LIN {X 0,Y 474.155,Z 514.396,A -85,B 0,C 180,E1 20492.017,E2 20492.017} C_VEL
LIN {X 0,Y 475.544,Z 517.886,A -85,B 0,C 180,E1 20491.079,E2 20491.079} C_VEL
LIN {X 0,Y 476.952,Z 519.954,A -85,B 0,C 180,E1 20490.456,E2 20490.456} C_VEL
LIN {X 0,Y 479.191,Z 523.963,A -85,B 0,C 180,E1 20489.394,E2 20489.394} C_VEL
LIN {X 0,Y 481.484,Z 528.373,A -85,B 0,C 180,E1 20488.305,E2 20488.305} C_VEL
LIN {X 0,Y 486.793,Z 538.934,A -85,B 0,C 180,E1 20485.892,E2 20485.892} C_VEL
LIN {X 0,Y 493.143,Z 551.884,A -85,B 0,C 180,E1 20483.213,E2 20483.213} C_VEL
LIN {X 0,Y 495.153,Z 556.027,A -85,B 0,C 180,E1 20482.476,E2 20482.476} C_VEL
LIN {X 0,Y 509.076,Z 575.515,A -85,B 0,C 180,E1 20480.277,E2 20480.277} C_VEL
LIN {X 0,Y 522.792,Z 596.581,A -85,B 0,C 180,E1 20478.273,E2 20478.273} C_VEL
LIN {X 0,Y 527.931,Z 605.432,A -85,B 0,C 180,E1 20477.547,E2 20477.547} C_VEL
LIN {X 0,Y 518.42,Z 845.443,A -85,B 0,C 180,E1 20473.808,E2 20473.808} C_VEL
LIN {X 0,Y 515.244,Z 924.905,A -85,B 0,C 180,E1 20472.535,E2 20472.535} C_VEL
LIN {X 0,Y 513.406,Z 949.561,A -85,B 0,C 180,E1 20471.961,E2 20471.961} C_VEL
LIN {X 0,Y 511.178,Z 973.065,A -85,B 0,C 180,E1 20471.232,E2 20471.232} C_VEL
LIN {X 0,Y 508.452,Z 995.949,A -85,B 0,C 180,E1 20470.313,E2 20470.313} C_VEL
LIN {X 0,Y 505.435,Z 1018.304,A -85,B 0,C 180,E1 20469.227,E2 20469.227} C_VEL
LIN {X 0,Y 502.044,Z 1040.134,A -85,B 0,C 180,E1 20467.936,E2 20467.936} C_VEL
LIN {X 0,Y 498.656,Z 1060.29,A -85,B 0,C 180,E1 20466.549,E2 20466.549} C_VEL
LIN {X 0,Y 494.89,Z 1080.931,A -85,B 0,C 180,E1 20464.873,E2 20464.873} C_VEL
LIN {X 0,Y 491.266,Z 1100.34,A -85,B 0,C 180,E1 20463.055,E2 20463.055} C_VEL
LIN {X 0,Y 487.78,Z 1118.193,A -85,B 0,C 180,E1 20461.101,E2 20461.101} C_VEL
LIN {X 0,Y 484.436,Z 1135.567,A -85,B 0,C 180,E1 20458.937,E2 20458.937} C_VEL
LIN {X 0,Y 481.445,Z 1151.258,A -85,B 0,C 180,E1 20456.653,E2 20456.653} C_VEL
LIN {X 0,Y 478.757,Z 1166.255,A -85,B 0,C 180,E1 20454.163,E2 20454.163} C_VEL
LIN {X 0,Y 476.612,Z 1179.063,A -85,B 0,C 180,E1 20451.662,E2 20451.662} C_VEL
LIN {X 0,Y 474.889,Z 1190.823,A -85,B 0,C 180,E1 20449.023,E2 20449.023} C_VEL
LIN {X 0,Y 473.606,Z 1200.885,A -85,B 0,C 180,E1 20446.307,E2 20446.307} C_VEL
LIN {X 0,Y 472.768,Z 1209.435,A -85,B 0,C 180,E1 20443.577,E2 20443.577} C_VEL
LIN {X 0,Y 472.242,Z 1216.419,A -85,B 0,C 180,E1 20440.738,E2 20440.738} C_VEL
LIN {X 0,Y 472.032,Z 1221.191,A -85,B 0,C 180,E1 20438.282,E2 20438.282} C_VEL
LIN {X 0,Y 471.92,Z 1225.242,A -85,B 0,C 180,E1 20435.349,E2 20435.349} C_VEL
LIN {X 0,Y 471.913,Z 1227.184,A -85,B 0,C 180,E1 20433.036,E2 20433.036} C_VEL
LIN {X 0,Y 471.916,Z 1228.071,A -85,B 0,C 180,E1 20430.728,E2 20430.728} C_VEL
LIN {X 0,Y 471.93,Z 1227.822,A -85,B 0,C 180,E1 20428.057,E2 20428.057} C_VEL
LIN {X 0,Y 471.933,Z 1225.961,A -85,B 0,C 180,E1 20425.382,E2 20425.382} C_VEL
LIN {X 0,Y 471.984,Z 1223.075,A -85,B 0,C 180,E1 20422.942,E2 20422.942} C_VEL
LIN {X 0,Y 472.159,Z 1218.019,A -85,B 0,C 180,E1 20420,E2 20420} C_VEL
LIN {X 0,Y 472.543,Z 1212,A -85,B 0,C 180,E1 20417.412,E2 20417.412} C_VEL
LIN {X 0,Y 473.256,Z 1204.234,A -85,B 0,C 180,E1 20414.687,E2 20414.687} C_VEL
LIN {X 0,Y 474.378,Z 1194.449,A -85,B 0,C 180,E1 20411.919,E2 20411.919} C_VEL
LIN {X 0,Y 475.903,Z 1183.735,A -85,B 0,C 180,E1 20409.331,E2 20409.331} C_VEL
LIN {X 0,Y 477.969,Z 1170.754,A -85,B 0,C 180,E1 20406.69,E2 20406.69} C_VEL
LIN {X 0,Y 480.439,Z 1156.789,A -85,B 0,C 180,E1 20404.218,E2 20404.218} C_VEL
LIN {X 0,Y 483.33,Z 1141.174,A -85,B 0,C 180,E1 20401.858,E2 20401.858} C_VEL
LIN {X 0,Y 486.577,Z 1124.421,A -85,B 0,C 180,E1 20399.635,E2 20399.635} C_VEL
LIN {X 0,Y 490.009,Z 1106.609,A -85,B 0,C 180,E1 20397.614,E2 20397.614} C_VEL
LIN {X 0,Y 493.65,Z 1087.708,A -85,B 0,C 180,E1 20395.732,E2 20395.732} C_VEL
LIN {X 0,Y 497.245,Z 1067.846,A -85,B 0,C 180,E1 20394.045,E2 20394.045} C_VEL
LIN {X 0,Y 500.924,Z 1046.802,A -85,B 0,C 180,E1 20392.498,E2 20392.498} C_VEL
LIN {X 0,Y 504.252,Z 1025.704,A -85,B 0,C 180,E1 20391.196,E2 20391.196} C_VEL
LIN {X 0,Y 507.471,Z 1003.563,A -85,B 0,C 180,E1 20390.036,E2 20390.036} C_VEL
LIN {X 0,Y 510.126,Z 981.826,A -85,B 0,C 180,E1 20389.107,E2 20389.107} C_VEL
LIN {X 0,Y 512.636,Z 958.481,A -85,B 0,C 180,E1 20388.297,E2 20388.297} C_VEL
LIN {X 0,Y 514.535,Z 935.049,A -85,B 0,C 180,E1 20387.69,E2 20387.69} C_VEL
LIN {X 0,Y 515.919,Z 910.67,A -85,B 0,C 180,E1 20387.223,E2 20387.223} C_VEL
LIN {X 0,Y 525.461,Z 664.98,A -85,B 0,C 180,E1 20383.375,E2 20383.375} C_VEL
LIN {X 0,Y 527.752,Z 604.829,A -85,B 0,C 180,E1 20382.433,E2 20382.433} C_VEL
LIN {X 0,Y 514.53,Z 583.673,A -85,B 0,C 180,E1 20380.552,E2 20380.552} C_VEL
LIN {X 0,Y 500.408,Z 563.192,A -85,B 0,C 180,E1 20378.402,E2 20378.402} C_VEL
LIN {X 0,Y 494.767,Z 555.412,A -85,B 0,C 180,E1 20377.467,E2 20377.467} C_VEL
LIN {X 0,Y 488.441,Z 542.064,A -85,B 0,C 180,E1 20374.829,E2 20374.829} C_VEL
LIN {X 0,Y 483.454,Z 532.413,A -85,B 0,C 180,E1 20372.671,E2 20372.671} C_VEL
LIN {X 0,Y 480.951,Z 527.653,A -85,B 0,C 180,E1 20371.531,E2 20371.531} C_VEL
LIN {X 0,Y 478.491,Z 523.082,A -85,B 0,C 180,E1 20370.378,E2 20370.378} C_VEL
LIN {X 0,Y 476.323,Z 518.832,A -85,B 0,C 180,E1 20369.282,E2 20369.282} C_VEL
LIN {X 0,Y 474.366,Z 515.411,A -85,B 0,C 180,E1 20368.312,E2 20368.312} C_VEL
LIN {X 0,Y 474.133,Z 514.262,A -85,B 0,C 180,E1 20367.916,E2 20367.916} C_VEL
LIN {X 0,Y 474.098,Z 514.151,A -85,B 0,C 180,E1 20364.284,E2 20364.284} C_VEL
LIN {X 0,Y 474.071,Z 514.151,A -85,B 0,C 180,E1 20360.753,E2 20360.753} C_VEL
LIN {X 0,Y 474.09,Z 514.148,A -85,B 0,C 180,E1 20357.174,E2 20357.174} C_VEL
LIN {X 0,Y 474.118,Z 514.152,A -85,B 0,C 180,E1 20353.663,E2 20353.663} C_VEL
LIN {X 0,Y 474.088,Z 514.176,A -85,B 0,C 180,E1 20350.082,E2 20350.082} C_VEL
LIN {X 0,Y 474.077,Z 514.166,A -85,B 0,C 180,E1 20346.418,E2 20346.418} C_VEL
LIN {X 0,Y 474.094,Z 514.146,A -85,B 0,C 180,E1 20342.78,E2 20342.78} C_VEL
LIN {X 0,Y 474.116,Z 514.142,A -85,B 0,C 180,E1 20339.275,E2 20339.275} C_VEL
LIN {X 0,Y 474.09,Z 514.163,A -85,B 0,C 180,E1 20335.645,E2 20335.645} C_VEL
LIN {X 0,Y 474.082,Z 514.178,A -85,B 0,C 180,E1 20331.998,E2 20331.998} C_VEL
LIN {X 0,Y 474.102,Z 514.154,A -85,B 0,C 180,E1 20328.442,E2 20328.442} C_VEL
LIN {X 0,Y 474.115,Z 514.143,A -85,B 0,C 180,E1 20324.84,E2 20324.84} C_VEL
LIN {X 0,Y 474.093,Z 514.147,A -85,B 0,C 180,E1 20321.251,E2 20321.251} C_VEL
LIN {X 0,Y 474.086,Z 514.154,A -85,B 0,C 180,E1 20317.689,E2 20317.689} C_VEL
LIN {X 0,Y 474.111,Z 514.156,A -85,B 0,C 180,E1 20314.115,E2 20314.115} C_VEL
LIN {X 0,Y 474.127,Z 514.429,A -85,B 0,C 180,E1 20311.467,E2 20311.467} C_VEL
LIN {X 0,Y 475.735,Z 518.072,A -85,B 0,C 180,E1 20310.471,E2 20310.471} C_VEL
LIN {X 0,Y 476.903,Z 519.937,A -85,B 0,C 180,E1 20309.927,E2 20309.927} C_VEL
LIN {X 0,Y 478.881,Z 523.608,A -85,B 0,C 180,E1 20308.954,E2 20308.954} C_VEL
LIN {X 0,Y 482.172,Z 530.174,A -85,B 0,C 180,E1 20307.341,E2 20307.341} C_VEL
LIN {X 0,Y 484.724,Z 535.255,A -85,B 0,C 180,E1 20306.154,E2 20306.154} C_VEL
LIN {X 0,Y 489.09,Z 544.038,A -85,B 0,C 180,E1 20304.218,E2 20304.218} C_VEL
LIN {X 0,Y 494.758,Z 556.102,A -85,B 0,C 180,E1 20301.799,E2 20301.799} C_VEL
LIN {X 0,Y 501.517,Z 571.621,A -85,B 0,C 180,E1 20299.009,E2 20299.009} C_VEL
LIN {X 0,Y 508.454,Z 589.192,A -85,B 0,C 180,E1 20296.194,E2 20296.194} C_VEL
LIN {X 0,Y 513.484,Z 603.577,A -85,B 0,C 180,E1 20294.117,E2 20294.117} C_VEL
LIN {X 0,Y 510.099,Z 627.117,A -85,B 0,C 180,E1 20292.145,E2 20292.145} C_VEL
LIN {X 0,Y 518.572,Z 680.793,A -85,B 0,C 180,E1 20290.232,E2 20290.232} C_VEL
LIN {X 0,Y 521.342,Z 700.88,A -85,B 0,C 180,E1 20289.597,E2 20289.597} C_VEL
LIN {X 0,Y 514.32,Z 951.65,A -85,B 0,C 180,E1 20286.124,E2 20286.124} C_VEL
LIN {X 0,Y 512.707,Z 973.976,A -85,B 0,C 180,E1 20285.653,E2 20285.653} C_VEL
LIN {X 0,Y 510.551,Z 995.541,A -85,B 0,C 180,E1 20285.016,E2 20285.016} C_VEL
LIN {X 0,Y 508.063,Z 1015.095,A -85,B 0,C 180,E1 20284.251,E2 20284.251} C_VEL
LIN {X 0,Y 504.852,Z 1036.457,A -85,B 0,C 180,E1 20283.203,E2 20283.203} C_VEL
LIN {X 0,Y 501.504,Z 1055.972,A -85,B 0,C 180,E1 20282.028,E2 20282.028} C_VEL
LIN {X 0,Y 497.867,Z 1074.515,A -85,B 0,C 180,E1 20280.671,E2 20280.671} C_VEL
LIN {X 0,Y 493.994,Z 1093.026,A -85,B 0,C 180,E1 20279.063,E2 20279.063} C_VEL
LIN {X 0,Y 490.378,Z 1109.28,A -85,B 0,C 180,E1 20277.39,E2 20277.39} C_VEL
LIN {X 0,Y 486.854,Z 1124.477,A -85,B 0,C 180,E1 20275.549,E2 20275.549} C_VEL
LIN {X 0,Y 486.127,Z 1127.636,A -85,B 0,C 180,E1 20275.13,E2 20275.13} C_VEL
LIN {X 0,Y 484.064,Z 1132.744,A -85,B 0,C 180,E1 20274.483,E2 20274.483} C_VEL
LIN {X 0,Y 475.596,Z 1145.16,A -85,B 0,C 180,E1 20272.883,E2 20272.883} C_VEL
LIN {X 0,Y 473.58,Z 1149.608,A -85,B 0,C 180,E1 20272.155,E2 20272.155} C_VEL
LIN {X 0,Y 470.739,Z 1161.868,A -85,B 0,C 180,E1 20269.784,E2 20269.784} C_VEL
LIN {X 0,Y 468.375,Z 1172.626,A -85,B 0,C 180,E1 20267.261,E2 20267.261} C_VEL
LIN {X 0,Y 466.516,Z 1182.255,A -85,B 0,C 180,E1 20264.522,E2 20264.522} C_VEL
LIN {X 0,Y 465.325,Z 1189.709,A -85,B 0,C 180,E1 20261.904,E2 20261.904} C_VEL
LIN {X 0,Y 464.56,Z 1195.655,A -85,B 0,C 180,E1 20259.164,E2 20259.164} C_VEL
LIN {X 0,Y 464.143,Z 1200.188,A -85,B 0,C 180,E1 20256.307,E2 20256.307} C_VEL
LIN {X 0,Y 464.002,Z 1202.847,A -85,B 0,C 180,E1 20253.707,E2 20253.707} C_VEL
LIN {X 0,Y 463.961,Z 1204.118,A -85,B 0,C 180,E1 20250.988,E2 20250.988} C_VEL
LIN {X 0,Y 463.962,Z 1204.008,A -85,B 0,C 180,E1 20248.271,E2 20248.271} C_VEL
LIN {X 0,Y 464.03,Z 1202.291,A -85,B 0,C 180,E1 20245.551,E2 20245.551} C_VEL
LIN {X 0,Y 464.238,Z 1198.967,A -85,B 0,C 180,E1 20242.7,E2 20242.7} C_VEL
LIN {X 0,Y 464.702,Z 1194.401,A -85,B 0,C 180,E1 20240.088,E2 20240.088} C_VEL
LIN {X 0,Y 465.569,Z 1187.959,A -85,B 0,C 180,E1 20237.346,E2 20237.346} C_VEL
LIN {X 0,Y 466.914,Z 1180.215,A -85,B 0,C 180,E1 20234.728,E2 20234.728} C_VEL
LIN {X 0,Y 468.827,Z 1170.537,A -85,B 0,C 180,E1 20232.115,E2 20232.115} C_VEL
LIN {X 0,Y 471.404,Z 1158.887,A -85,B 0,C 180,E1 20229.515,E2 20229.515} C_VEL
LIN {X 0,Y 474.37,Z 1146.429,A -85,B 0,C 180,E1 20227.181,E2 20227.181} C_VEL
LIN {X 0,Y 477.553,Z 1133.278,A -85,B 0,C 180,E1 20225.113,E2 20225.113} C_VEL
LIN {X 0,Y 481.473,Z 1117.091,A -85,B 0,C 180,E1 20222.949,E2 20222.949} C_VEL
LIN {X 0,Y 485.362,Z 1100.85,A -85,B 0,C 180,E1 20221.109,E2 20221.109} C_VEL
LIN {X 0,Y 489.163,Z 1083.804,A -85,B 0,C 180,E1 20219.491,E2 20219.491} C_VEL
LIN {X 0,Y 493.259,Z 1064.206,A -85,B 0,C 180,E1 20217.921,E2 20217.921} C_VEL
LIN {X 0,Y 496.963,Z 1044.87,A -85,B 0,C 180,E1 20216.634,E2 20216.634} C_VEL
LIN {X 0,Y 500.265,Z 1024.901,A -85,B 0,C 180,E1 20215.555,E2 20215.555} C_VEL
LIN {X 0,Y 503.312,Z 1003.371,A -85,B 0,C 180,E1 20214.614,E2 20214.614} C_VEL
LIN {X 0,Y 505.699,Z 982.724,A -85,B 0,C 180,E1 20213.917,E2 20213.917} C_VEL
LIN {X 0,Y 507.619,Z 960.502,A -85,B 0,C 180,E1 20213.375,E2 20213.375} C_VEL
LIN {X 0,Y 508.783,Z 936.875,A -85,B 0,C 180,E1 20212.979,E2 20212.979} C_VEL
LIN {X 0,Y 515.475,Z 700.609,A -85,B 0,C 180,E1 20209.68,E2 20209.68} C_VEL
LIN {X 0,Y 507.716,Z 648.72,A -85,B 0,C 180,E1 20207.879,E2 20207.879} C_VEL
LIN {X 0,Y 504.105,Z 625.337,A -85,B 0,C 180,E1 20206.976,E2 20206.976} C_VEL
LIN {X 0,Y 506.962,Z 606.936,A -85,B 0,C 180,E1 20205.399,E2 20205.399} C_VEL
LIN {X 0,Y 500.415,Z 588.775,A -85,B 0,C 180,E1 20202.669,E2 20202.669} C_VEL
LIN {X 0,Y 493.848,Z 572.457,A -85,B 0,C 180,E1 20199.929,E2 20199.929} C_VEL
LIN {X 0,Y 487.537,Z 558.088,A -85,B 0,C 180,E1 20197.23,E2 20197.23} C_VEL
LIN {X 0,Y 482.013,Z 546.324,A -85,B 0,C 180,E1 20194.771,E2 20194.771} C_VEL
LIN {X 0,Y 477.796,Z 537.861,A -85,B 0,C 180,E1 20192.821,E2 20192.821} C_VEL
LIN {X 0,Y 475.073,Z 532.675,A -85,B 0,C 180,E1 20191.529,E2 20191.529} C_VEL
LIN {X 0,Y 473.555,Z 529.451,A -85,B 0,C 180,E1 20190.729,E2 20190.729} C_VEL
LIN {X 0,Y 471.63,Z 525.759,A -85,B 0,C 180,E1 20189.742,E2 20189.742} C_VEL
LIN {X 0,Y 469.026,Z 521.007,A -85,B 0,C 180,E1 20188.386,E2 20188.386} C_VEL
LIN {X 0,Y 466.326,Z 516.083,A -85,B 0,C 180,E1 20186.881,E2 20186.881} C_VEL
LIN {X 0,Y 466.157,Z 515.237,A -85,B 0,C 180,E1 20186.497,E2 20186.497} C_VEL
LIN {X 0,Y 466.147,Z 515.137,A -85,B 0,C 180,E1 20182.732,E2 20182.732} C_VEL
LIN {X 0,Y 466.173,Z 515.132,A -85,B 0,C 180,E1 20179.158,E2 20179.158} C_VEL
LIN {X 0,Y 466.171,Z 515.136,A -85,B 0,C 180,E1 20175.552,E2 20175.552} C_VEL
LIN {X 0,Y 466.142,Z 515.158,A -85,B 0,C 180,E1 20172.009,E2 20172.009} C_VEL
LIN {X 0,Y 466.144,Z 515.166,A -85,B 0,C 180,E1 20168.263,E2 20168.263} C_VEL
LIN {X 0,Y 466.166,Z 515.14,A -85,B 0,C 180,E1 20164.675,E2 20164.675} C_VEL
LIN {X 0,Y 466.173,Z 515.129,A -85,B 0,C 180,E1 20160.983,E2 20160.983} C_VEL
LIN {X 0,Y 466.14,Z 515.141,A -85,B 0,C 180,E1 20157.418,E2 20157.418} C_VEL
LIN {X 0,Y 466.139,Z 515.162,A -85,B 0,C 180,E1 20153.719,E2 20153.719} C_VEL
LIN {X 0,Y 466.159,Z 515.157,A -85,B 0,C 180,E1 20150.119,E2 20150.119} C_VEL
LIN {X 0,Y 466.177,Z 515.137,A -85,B 0,C 180,E1 20146.48,E2 20146.48} C_VEL
LIN {X 0,Y 466.141,Z 515.135,A -85,B 0,C 180,E1 20142.91,E2 20142.91} C_VEL
LIN {X 0,Y 466.131,Z 515.138,A -85,B 0,C 180,E1 20139.264,E2 20139.264} C_VEL
LIN {X 0,Y 466.155,Z 515.139,A -85,B 0,C 180,E1 20135.68,E2 20135.68} C_VEL
LIN {X 0,Y 466.204,Z 515.444,A -85,B 0,C 180,E1 20133.681,E2 20133.681} C_VEL
LIN {X 0,Y 467.491,Z 518.71,A -85,B 0,C 180,E1 20132.76,E2 20132.76} C_VEL
LIN {X 0,Y 469.06,Z 520.891,A -85,B 0,C 180,E1 20132.032,E2 20132.032} C_VEL
LIN {X 0,Y 470.968,Z 524.611,A -85,B 0,C 180,E1 20131.006,E2 20131.006} C_VEL
LIN {X 0,Y 472.301,Z 527.272,A -85,B 0,C 180,E1 20130.304,E2 20130.304} C_VEL
LIN {X 0,Y 474.398,Z 531.003,A -85,B 0,C 180,E1 20129.307,E2 20129.307} C_VEL
LIN {X 0,Y 477.153,Z 536.384,A -85,B 0,C 180,E1 20127.983,E2 20127.983} C_VEL
LIN {X 0,Y 481.197,Z 544.202,A -85,B 0,C 180,E1 20126.159,E2 20126.159} C_VEL
LIN {X 0,Y 487.509,Z 557.043,A -85,B 0,C 180,E1 20123.502,E2 20123.502} C_VEL
LIN {X 0,Y 501.063,Z 575.927,A -85,B 0,C 180,E1 20121.255,E2 20121.255} C_VEL
LIN {X 0,Y 513.716,Z 594.998,A -85,B 0,C 180,E1 20119.323,E2 20119.323} C_VEL
LIN {X 0,Y 522.067,Z 608.776,A -85,B 0,C 180,E1 20118.108,E2 20118.108} C_VEL
LIN {X 0,Y 512.25,Z 848.274,A -85,B 0,C 180,E1 20114.346,E2 20114.346} C_VEL
LIN {X 0,Y 509.051,Z 925.38,A -85,B 0,C 180,E1 20113.099,E2 20113.099} C_VEL
LIN {X 0,Y 507.158,Z 949.918,A -85,B 0,C 180,E1 20112.522,E2 20112.522} C_VEL
LIN {X 0,Y 504.866,Z 973.275,A -85,B 0,C 180,E1 20111.791,E2 20111.791} C_VEL
LIN {X 0,Y 502.065,Z 996.036,A -85,B 0,C 180,E1 20110.87,E2 20110.87} C_VEL
LIN {X 0,Y 498.862,Z 1018.969,A -85,B 0,C 180,E1 20109.744,E2 20109.744} C_VEL
LIN {X 0,Y 495.344,Z 1040.705,A -85,B 0,C 180,E1 20108.44,E2 20108.44} C_VEL
LIN {X 0,Y 491.751,Z 1061.312,A -85,B 0,C 180,E1 20107.002,E2 20107.002} C_VEL
LIN {X 0,Y 487.845,Z 1081.773,A -85,B 0,C 180,E1 20105.308,E2 20105.308} C_VEL
LIN {X 0,Y 483.989,Z 1101.508,A -85,B 0,C 180,E1 20103.421,E2 20103.421} C_VEL
LIN {X 0,Y 480.46,Z 1118.817,A -85,B 0,C 180,E1 20101.489,E2 20101.489} C_VEL
LIN {X 0,Y 476.999,Z 1136.02,A -85,B 0,C 180,E1 20099.305,E2 20099.305} C_VEL
LIN {X 0,Y 473.864,Z 1151.706,A -85,B 0,C 180,E1 20096.978,E2 20096.978} C_VEL
LIN {X 0,Y 471.06,Z 1166.601,A -85,B 0,C 180,E1 20094.45,E2 20094.45} C_VEL
LIN {X 0,Y 468.825,Z 1179.341,A -85,B 0,C 180,E1 20091.912,E2 20091.912} C_VEL
LIN {X 0,Y 466.954,Z 1191.423,A -85,B 0,C 180,E1 20089.124,E2 20089.124} C_VEL
LIN {X 0,Y 465.674,Z 1201.048,A -85,B 0,C 180,E1 20086.464,E2 20086.464} C_VEL
LIN {X 0,Y 464.796,Z 1209.535,A -85,B 0,C 180,E1 20083.688,E2 20083.688} C_VEL
LIN {X 0,Y 464.261,Z 1216.335,A -85,B 0,C 180,E1 20080.856,E2 20080.856} C_VEL
LIN {X 0,Y 464.035,Z 1221.186,A -85,B 0,C 180,E1 20078.3,E2 20078.3} C_VEL
LIN {X 0,Y 463.924,Z 1225.031,A -85,B 0,C 180,E1 20075.441,E2 20075.441} C_VEL
LIN {X 0,Y 463.916,Z 1226.978,A -85,B 0,C 180,E1 20073.089,E2 20073.089} C_VEL
LIN {X 0,Y 463.919,Z 1227.866,A -85,B 0,C 180,E1 20070.741,E2 20070.741} C_VEL
LIN {X 0,Y 463.933,Z 1227.617,A -85,B 0,C 180,E1 20068.024,E2 20068.024} C_VEL
LIN {X 0,Y 463.931,Z 1225.75,A -85,B 0,C 180,E1 20065.302,E2 20065.302} C_VEL
LIN {X 0,Y 463.985,Z 1223.027,A -85,B 0,C 180,E1 20062.944,E2 20062.944} C_VEL
LIN {X 0,Y 464.155,Z 1218.322,A -85,B 0,C 180,E1 20060.077,E2 20060.077} C_VEL
LIN {X 0,Y 464.563,Z 1212.076,A -85,B 0,C 180,E1 20057.319,E2 20057.319} C_VEL
LIN {X 0,Y 465.263,Z 1204.723,A -85,B 0,C 180,E1 20054.673,E2 20054.673} C_VEL
LIN {X 0,Y 466.404,Z 1195.252,A -85,B 0,C 180,E1 20051.89,E2 20051.89} C_VEL
LIN {X 0,Y 467.871,Z 1185.251,A -85,B 0,C 180,E1 20049.4,E2 20049.4} C_VEL
LIN {X 0,Y 470.103,Z 1171.867,A -85,B 0,C 180,E1 20046.564,E2 20046.564} C_VEL
LIN {X 0,Y 472.378,Z 1159.368,A -85,B 0,C 180,E1 20044.284,E2 20044.284} C_VEL
LIN {X 0,Y 475.658,Z 1142.549,A -85,B 0,C 180,E1 20041.637,E2 20041.637} C_VEL
LIN {X 0,Y 478.798,Z 1126.91,A -85,B 0,C 180,E1 20039.506,E2 20039.506} C_VEL
LIN {X 0,Y 482.55,Z 1108.439,A -85,B 0,C 180,E1 20037.333,E2 20037.333} C_VEL
LIN {X 0,Y 486.038,Z 1091.007,A -85,B 0,C 180,E1 20035.548,E2 20035.548} C_VEL
LIN {X 0,Y 490.049,Z 1070.067,A -85,B 0,C 180,E1 20033.703,E2 20033.703} C_VEL
LIN {X 0,Y 493.756,Z 1049.73,A -85,B 0,C 180,E1 20032.165,E2 20032.165} C_VEL
LIN {X 0,Y 497.354,Z 1028.058,A -85,B 0,C 180,E1 20030.783,E2 20030.783} C_VEL
LIN {X 0,Y 500.502,Z 1007.339,A -85,B 0,C 180,E1 20029.665,E2 20029.665} C_VEL
LIN {X 0,Y 503.594,Z 983.594,A -85,B 0,C 180,E1 20028.612,E2 20028.612} C_VEL
LIN {X 0,Y 506.006,Z 961.948,A -85,B 0,C 180,E1 20027.839,E2 20027.839} C_VEL
LIN {X 0,Y 508.183,Z 937.31,A -85,B 0,C 180,E1 20027.169,E2 20027.169} C_VEL
LIN {X 0,Y 509.549,Z 915.033,A -85,B 0,C 180,E1 20026.725,E2 20026.725} C_VEL
LIN {X 0,Y 519.396,Z 671.122,A -85,B 0,C 180,E1 20022.865,E2 20022.865} C_VEL
LIN {X 0,Y 521.884,Z 608.216,A -85,B 0,C 180,E1 20021.872,E2 20021.872} C_VEL
LIN {X 0,Y 508.399,Z 586.776,A -85,B 0,C 180,E1 20019.897,E2 20019.897} C_VEL
LIN {X 0,Y 494.504,Z 566.61,A -85,B 0,C 180,E1 20017.71,E2 20017.71} C_VEL
LIN {X 0,Y 487.167,Z 556.44,A -85,B 0,C 180,E1 20016.435,E2 20016.435} C_VEL
LIN {X 0,Y 480.604,Z 542.941,A -85,B 0,C 180,E1 20013.601,E2 20013.601} C_VEL
LIN {X 0,Y 475.803,Z 533.692,A -85,B 0,C 180,E1 20011.411,E2 20011.411} C_VEL
LIN {X 0,Y 473.231,Z 528.939,A -85,B 0,C 180,E1 20010.19,E2 20010.19} C_VEL
LIN {X 0,Y 471.072,Z 524.729,A -85,B 0,C 180,E1 20009.083,E2 20009.083} C_VEL
LIN {X 0,Y 469.122,Z 521.117,A -85,B 0,C 180,E1 20008.07,E2 20008.07} C_VEL
LIN {X 0,Y 468.152,Z 519.517,A -85,B 0,C 180,E1 20007.584,E2 20007.584} C_VEL
LIN {X 0,Y 466.386,Z 516.358,A -85,B 0,C 180,E1 20006.621,E2 20006.621} C_VEL
LIN {X 0,Y 466.18,Z 515.248,A -85,B 0,C 180,E1 20006.222,E2 20006.222} C_VEL
LIN {X 0,Y 466.137,Z 515.165,A -85,B 0,C 180,E1 20002.713,E2 20002.713} C_VEL
LIN {X 0,Y 466.143,Z 515.168,A -85,B 0,C 180,E1 19999.029,E2 19999.029} C_VEL
LIN {X 0,Y 466.179,Z 515.15,A -85,B 0,C 180,E1 19995.424,E2 19995.424} C_VEL
LIN {X 0,Y 466.167,Z 515.136,A -85,B 0,C 180,E1 19991.757,E2 19991.757} C_VEL
LIN {X 0,Y 466.139,Z 515.13,A -85,B 0,C 180,E1 19988.139,E2 19988.139} C_VEL
LIN {X 0,Y 466.139,Z 515.138,A -85,B 0,C 180,E1 19984.429,E2 19984.429} C_VEL
LIN {X 0,Y 466.162,Z 515.159,A -85,B 0,C 180,E1 19980.737,E2 19980.737} C_VEL
LIN {X 0,Y 466.175,Z 515.157,A -85,B 0,C 180,E1 19977.049,E2 19977.049} C_VEL
LIN {X 0,Y 466.167,Z 515.136,A -85,B 0,C 180,E1 19973.349,E2 19973.349} C_VEL
LIN {X 0,Y 466.142,Z 515.133,A -85,B 0,C 180,E1 19969.744,E2 19969.744} C_VEL
LIN {X 0,Y 466.152,Z 515.14,A -85,B 0,C 180,E1 19966.099,E2 19966.099} C_VEL
LIN {X 0,Y 466.177,Z 515.154,A -85,B 0,C 180,E1 19962.525,E2 19962.525} C_VEL
LIN {X 0,Y 466.175,Z 515.164,A -85,B 0,C 180,E1 19958.879,E2 19958.879} C_VEL
LIN {X 0,Y 466.149,Z 515.163,A -85,B 0,C 180,E1 19955.274,E2 19955.274} C_VEL
LIN {X 0,Y 466.197,Z 515.449,A -85,B 0,C 180,E1 19953.151,E2 19953.151} C_VEL
LIN {X 0,Y 467.784,Z 519.045,A -85,B 0,C 180,E1 19952.088,E2 19952.088} C_VEL
LIN {X 0,Y 469.02,Z 520.979,A -85,B 0,C 180,E1 19951.475,E2 19951.475} C_VEL
LIN {X 0,Y 471.172,Z 524.818,A -85,B 0,C 180,E1 19950.366,E2 19950.366} C_VEL
LIN {X 0,Y 473.564,Z 529.455,A -85,B 0,C 180,E1 19949.131,E2 19949.131} C_VEL
LIN {X 0,Y 478.643,Z 539.359,A -85,B 0,C 180,E1 19946.673,E2 19946.673} C_VEL
LIN {X 0,Y 485.077,Z 552.741,A -85,B 0,C 180,E1 19943.73,E2 19943.73} C_VEL
LIN {X 0,Y 491.581,Z 567.183,A -85,B 0,C 180,E1 19940.909,E2 19940.909} C_VEL
LIN {X 0,Y 498.329,Z 583.494,A -85,B 0,C 180,E1 19938.075,E2 19938.075} C_VEL
LIN {X 0,Y 505.021,Z 601.388,A -85,B 0,C 180,E1 19935.297,E2 19935.297} C_VEL
LIN {X 0,Y 506.908,Z 606.859,A -85,B 0,C 180,E1 19934.506,E2 19934.506} C_VEL
LIN {X 0,Y 504.045,Z 626.234,A -85,B 0,C 180,E1 19932.87,E2 19932.87} C_VEL
LIN {X 0,Y 512.128,Z 678.026,A -85,B 0,C 180,E1 19930.975,E2 19930.975} C_VEL
LIN {X 0,Y 515.471,Z 702.355,A -85,B 0,C 180,E1 19930.185,E2 19930.185} C_VEL
LIN {X 0,Y 508.157,Z 951.353,A -85,B 0,C 180,E1 19926.7,E2 19926.7} C_VEL
LIN {X 0,Y 506.503,Z 973.594,A -85,B 0,C 180,E1 19926.229,E2 19926.229} C_VEL
LIN {X 0,Y 504.374,Z 994.496,A -85,B 0,C 180,E1 19925.614,E2 19925.614} C_VEL
LIN {X 0,Y 501.603,Z 1015.5,A -85,B 0,C 180,E1 19924.787,E2 19924.787} C_VEL
LIN {X 0,Y 498.256,Z 1036.893,A -85,B 0,C 180,E1 19923.723,E2 19923.723} C_VEL
LIN {X 0,Y 494.75,Z 1056.62,A -85,B 0,C 180,E1 19922.518,E2 19922.518} C_VEL
LIN {X 0,Y 490.991,Z 1075.05,A -85,B 0,C 180,E1 19921.148,E2 19921.148} C_VEL
LIN {X 0,Y 486.978,Z 1093.469,A -85,B 0,C 180,E1 19919.522,E2 19919.522} C_VEL
LIN {X 0,Y 483.176,Z 1109.95,A -85,B 0,C 180,E1 19917.801,E2 19917.801} C_VEL
LIN {X 0,Y 479.356,Z 1125.728,A -85,B 0,C 180,E1 19915.845,E2 19915.845} C_VEL
LIN {X 0,Y 475.927,Z 1139.912,A -85,B 0,C 180,E1 19913.789,E2 19913.789} C_VEL
LIN {X 0,Y 473.58,Z 1149.608,A -85,B 0,C 180,E1 19912.155,E2 19912.155} C_VEL
LIN {X 0,Y 471.604,Z 1154.028,A -85,B 0,C 180,E1 19911.407,E2 19911.407} C_VEL
LIN {X 0,Y 463.475,Z 1164.458,A -85,B 0,C 180,E1 19909.551,E2 19909.551} C_VEL
LIN {X 0,Y 461.698,Z 1168.191,A -85,B 0,C 180,E1 19908.743,E2 19908.743} C_VEL
LIN {X 0,Y 459.564,Z 1177.934,A -85,B 0,C 180,E1 19906.17,E2 19906.17} C_VEL
LIN {X 0,Y 457.944,Z 1186.584,A -85,B 0,C 180,E1 19903.382,E2 19903.382} C_VEL
LIN {X 0,Y 456.948,Z 1193.11,A -85,B 0,C 180,E1 19900.719,E2 19900.719} C_VEL
LIN {X 0,Y 456.344,Z 1198.249,A -85,B 0,C 180,E1 19897.934,E2 19897.934} C_VEL
LIN {X 0,Y 456.069,Z 1201.882,A -85,B 0,C 180,E1 19895.157,E2 19895.157} C_VEL
LIN {X 0,Y 455.978,Z 1203.86,A -85,B 0,C 180,E1 19892.388,E2 19892.388} C_VEL
LIN {X 0,Y 455.955,Z 1204.424,A -85,B 0,C 180,E1 19889.497,E2 19889.497} C_VEL
LIN {X 0,Y 455.988,Z 1203.528,A -85,B 0,C 180,E1 19886.858,E2 19886.858} C_VEL
LIN {X 0,Y 456.122,Z 1200.966,A -85,B 0,C 180,E1 19883.96,E2 19883.96} C_VEL
LIN {X 0,Y 456.488,Z 1197.021,A -85,B 0,C 180,E1 19881.18,E2 19881.18} C_VEL
LIN {X 0,Y 457.2,Z 1191.321,A -85,B 0,C 180,E1 19878.393,E2 19878.393} C_VEL
LIN {X 0,Y 458.487,Z 1183.56,A -85,B 0,C 180,E1 19875.476,E2 19875.476} C_VEL
LIN {X 0,Y 460.268,Z 1174.731,A -85,B 0,C 180,E1 19872.816,E2 19872.816} C_VEL
LIN {X 0,Y 462.567,Z 1164.411,A -85,B 0,C 180,E1 19870.294,E2 19870.294} C_VEL
LIN {X 0,Y 465.552,Z 1152.084,A -85,B 0,C 180,E1 19867.772,E2 19867.772} C_VEL
LIN {X 0,Y 468.993,Z 1138.508,A -85,B 0,C 180,E1 19865.435,E2 19865.435} C_VEL
LIN {X 0,Y 472.647,Z 1124.053,A -85,B 0,C 180,E1 19863.354,E2 19863.354} C_VEL
LIN {X 0,Y 476.825,Z 1107.25,A -85,B 0,C 180,E1 19861.302,E2 19861.302} C_VEL
LIN {X 0,Y 480.844,Z 1090.624,A -85,B 0,C 180,E1 19859.58,E2 19859.58} C_VEL
LIN {X 0,Y 484.749,Z 1073.043,A -85,B 0,C 180,E1 19858.058,E2 19858.058} C_VEL
LIN {X 0,Y 488.655,Z 1054.163,A -85,B 0,C 180,E1 19856.675,E2 19856.675} C_VEL
LIN {X 0,Y 492.092,Z 1035.425,A -85,B 0,C 180,E1 19855.537,E2 19855.537} C_VEL
LIN {X 0,Y 495.364,Z 1015.075,A -85,B 0,C 180,E1 19854.529,E2 19854.529} C_VEL
LIN {X 0,Y 498.22,Z 994.116,A -85,B 0,C 180,E1 19853.699,E2 19853.699} C_VEL
LIN {X 0,Y 500.452,Z 972.815,A -85,B 0,C 180,E1 19853.072,E2 19853.072} C_VEL
LIN {X 0,Y 502.159,Z 949.965,A -85,B 0,C 180,E1 19852.593,E2 19852.593} C_VEL
LIN {X 0,Y 509.687,Z 702.178,A -85,B 0,C 180,E1 19849.083,E2 19849.083} C_VEL
LIN {X 0,Y 502.03,Z 649.959,A -85,B 0,C 180,E1 19847.235,E2 19847.235} C_VEL
LIN {X 0,Y 498.128,Z 624.609,A -85,B 0,C 180,E1 19846.244,E2 19846.244} C_VEL
LIN {X 0,Y 500.37,Z 610.512,A -85,B 0,C 180,E1 19845.024,E2 19845.024} C_VEL
LIN {X 0,Y 494.157,Z 593.11,A -85,B 0,C 180,E1 19842.361,E2 19842.361} C_VEL
LIN {X 0,Y 487.628,Z 576.713,A -85,B 0,C 180,E1 19839.559,E2 19839.559} C_VEL
LIN {X 0,Y 481.52,Z 562.728,A -85,B 0,C 180,E1 19836.879,E2 19836.879} C_VEL
LIN {X 0,Y 476.017,Z 550.946,A -85,B 0,C 180,E1 19834.363,E2 19834.363} C_VEL
LIN {X 0,Y 470.741,Z 540.046,A -85,B 0,C 180,E1 19831.788,E2 19831.788} C_VEL
LIN {X 0,Y 467.697,Z 534.485,A -85,B 0,C 180,E1 19830.301,E2 19830.301} C_VEL
LIN {X 0,Y 465.608,Z 530.334,A -85,B 0,C 180,E1 19829.175,E2 19829.175} C_VEL
LIN {X 0,Y 463.096,Z 525.617,A -85,B 0,C 180,E1 19827.799,E2 19827.799} C_VEL
LIN {X 0,Y 461.136,Z 521.934,A -85,B 0,C 180,E1 19826.67,E2 19826.67} C_VEL
LIN {X 0,Y 458.395,Z 517.091,A -85,B 0,C 180,E1 19825.035,E2 19825.035} C_VEL
LIN {X 0,Y 458.215,Z 516.214,A -85,B 0,C 180,E1 19824.632,E2 19824.632} C_VEL
LIN {X 0,Y 458.226,Z 516.153,A -85,B 0,C 180,E1 19820.949,E2 19820.949} C_VEL
LIN {X 0,Y 458.239,Z 516.144,A -85,B 0,C 180,E1 19817.263,E2 19817.263} C_VEL
LIN {X 0,Y 458.232,Z 516.132,A -85,B 0,C 180,E1 19813.502,E2 19813.502} C_VEL
LIN {X 0,Y 458.205,Z 516.123,A -85,B 0,C 180,E1 19809.8,E2 19809.8} C_VEL
LIN {X 0,Y 458.199,Z 516.122,A -85,B 0,C 180,E1 19806.138,E2 19806.138} C_VEL
LIN {X 0,Y 458.22,Z 516.135,A -85,B 0,C 180,E1 19802.501,E2 19802.501} C_VEL
LIN {X 0,Y 458.241,Z 516.153,A -85,B 0,C 180,E1 19798.875,E2 19798.875} C_VEL
LIN {X 0,Y 458.215,Z 516.135,A -85,B 0,C 180,E1 19795.118,E2 19795.118} C_VEL
LIN {X 0,Y 458.191,Z 516.122,A -85,B 0,C 180,E1 19791.593,E2 19791.593} C_VEL
LIN {X 0,Y 458.215,Z 516.124,A -85,B 0,C 180,E1 19788.036,E2 19788.036} C_VEL
LIN {X 0,Y 458.244,Z 516.134,A -85,B 0,C 180,E1 19784.432,E2 19784.432} C_VEL
LIN {X 0,Y 458.213,Z 516.15,A -85,B 0,C 180,E1 19780.761,E2 19780.761} C_VEL
LIN {X 0,Y 458.194,Z 516.156,A -85,B 0,C 180,E1 19777.142,E2 19777.142} C_VEL
LIN {X 0,Y 458.258,Z 516.481,A -85,B 0,C 180,E1 19775.531,E2 19775.531} C_VEL
LIN {X 0,Y 459.675,Z 519.837,A -85,B 0,C 180,E1 19774.488,E2 19774.488} C_VEL
LIN {X 0,Y 461.146,Z 521.871,A -85,B 0,C 180,E1 19773.747,E2 19773.747} C_VEL
LIN {X 0,Y 463.102,Z 525.636,A -85,B 0,C 180,E1 19772.62,E2 19772.62} C_VEL
LIN {X 0,Y 464.052,Z 527.265,A -85,B 0,C 180,E1 19772.123,E2 19772.123} C_VEL
LIN {X 0,Y 466.862,Z 532.602,A -85,B 0,C 180,E1 19770.629,E2 19770.629} C_VEL
LIN {X 0,Y 469.319,Z 537.289,A -85,B 0,C 180,E1 19769.39,E2 19769.39} C_VEL
LIN {X 0,Y 471.86,Z 542.221,A -85,B 0,C 180,E1 19768.154,E2 19768.154} C_VEL
LIN {X 0,Y 476.093,Z 550.656,A -85,B 0,C 180,E1 19766.182,E2 19766.182} C_VEL
LIN {X 0,Y 479.907,Z 558.307,A -85,B 0,C 180,E1 19764.568,E2 19764.568} C_VEL
LIN {X 0,Y 492.546,Z 575.495,A -85,B 0,C 180,E1 19762.372,E2 19762.372} C_VEL
LIN {X 0,Y 506.218,Z 595.701,A -85,B 0,C 180,E1 19760.192,E2 19760.192} C_VEL
LIN {X 0,Y 516.258,Z 612.041,A -85,B 0,C 180,E1 19758.684,E2 19758.684} C_VEL
LIN {X 0,Y 506.127,Z 851.124,A -85,B 0,C 180,E1 19754.898,E2 19754.898} C_VEL
LIN {X 0,Y 502.917,Z 925.749,A -85,B 0,C 180,E1 19753.679,E2 19753.679} C_VEL
LIN {X 0,Y 500.966,Z 950.215,A -85,B 0,C 180,E1 19753.098,E2 19753.098} C_VEL
LIN {X 0,Y 498.594,Z 973.605,A -85,B 0,C 180,E1 19752.361,E2 19752.361} C_VEL
LIN {X 0,Y 495.677,Z 996.511,A -85,B 0,C 180,E1 19751.424,E2 19751.424} C_VEL
LIN {X 0,Y 492.389,Z 1019.228,A -85,B 0,C 180,E1 19750.297,E2 19750.297} C_VEL
LIN {X 0,Y 488.905,Z 1040.01,A -85,B 0,C 180,E1 19749.042,E2 19749.042} C_VEL
LIN {X 0,Y 485.176,Z 1060.687,A -85,B 0,C 180,E1 19747.589,E2 19747.589} C_VEL
LIN {X 0,Y 481.109,Z 1081.253,A -85,B 0,C 180,E1 19745.878,E2 19745.878} C_VEL
LIN {X 0,Y 477.172,Z 1100.614,A -85,B 0,C 180,E1 19744.019,E2 19744.019} C_VEL
LIN {X 0,Y 473.271,Z 1118.925,A -85,B 0,C 180,E1 19741.953,E2 19741.953} C_VEL
LIN {X 0,Y 469.667,Z 1136.099,A -85,B 0,C 180,E1 19739.737,E2 19739.737} C_VEL
LIN {X 0,Y 466.459,Z 1151.362,A -85,B 0,C 180,E1 19737.442,E2 19737.442} C_VEL
LIN {X 0,Y 463.65,Z 1165.621,A -85,B 0,C 180,E1 19735.003,E2 19735.003} C_VEL
LIN {X 0,Y 461.251,Z 1178.44,A -85,B 0,C 180,E1 19732.428,E2 19732.428} C_VEL
LIN {X 0,Y 459.31,Z 1190.168,A -85,B 0,C 180,E1 19729.719,E2 19729.719} C_VEL
LIN {X 0,Y 457.849,Z 1200.365,A -85,B 0,C 180,E1 19726.885,E2 19726.885} C_VEL
LIN {X 0,Y 456.918,Z 1208.568,A -85,B 0,C 180,E1 19724.187,E2 19724.187} C_VEL
LIN {X 0,Y 456.312,Z 1215.691,A -85,B 0,C 180,E1 19721.246,E2 19721.246} C_VEL
LIN {X 0,Y 456.063,Z 1220.53,A -85,B 0,C 180,E1 19718.701,E2 19718.701} C_VEL
LIN {X 0,Y 455.934,Z 1224.701,A -85,B 0,C 180,E1 19715.663,E2 19715.663} C_VEL
LIN {X 0,Y 455.919,Z 1226.772,A -85,B 0,C 180,E1 19713.143,E2 19713.143} C_VEL
LIN {X 0,Y 455.922,Z 1227.662,A -85,B 0,C 180,E1 19710.754,E2 19710.754} C_VEL
LIN {X 0,Y 455.935,Z 1227.411,A -85,B 0,C 180,E1 19707.989,E2 19707.989} C_VEL
LIN {X 0,Y 455.929,Z 1225.54,A -85,B 0,C 180,E1 19705.22,E2 19705.22} C_VEL
LIN {X 0,Y 455.98,Z 1222.811,A -85,B 0,C 180,E1 19702.82,E2 19702.82} C_VEL
LIN {X 0,Y 456.168,Z 1218.093,A -85,B 0,C 180,E1 19699.901,E2 19699.901} C_VEL
LIN {X 0,Y 456.609,Z 1211.837,A -85,B 0,C 180,E1 19697.094,E2 19697.094} C_VEL
LIN {X 0,Y 457.358,Z 1204.473,A -85,B 0,C 180,E1 19694.401,E2 19694.401} C_VEL
LIN {X 0,Y 458.601,Z 1194.798,A -85,B 0,C 180,E1 19691.521,E2 19691.521} C_VEL
LIN {X 0,Y 460.158,Z 1184.774,A -85,B 0,C 180,E1 19688.991,E2 19688.991} C_VEL
LIN {X 0,Y 462.517,Z 1171.427,A -85,B 0,C 180,E1 19686.13,E2 19686.13} C_VEL
LIN {X 0,Y 464.9,Z 1159.038,A -85,B 0,C 180,E1 19683.839,E2 19683.839} C_VEL
LIN {X 0,Y 468.171,Z 1143.053,A -85,B 0,C 180,E1 19681.28,E2 19681.28} C_VEL
LIN {X 0,Y 471.435,Z 1127.476,A -85,B 0,C 180,E1 19679.119,E2 19679.119} C_VEL
LIN {X 0,Y 475.455,Z 1108.559,A -85,B 0,C 180,E1 19676.855,E2 19676.855} C_VEL
LIN {X 0,Y 479.085,Z 1091.147,A -85,B 0,C 180,E1 19675.048,E2 19675.048} C_VEL
LIN {X 0,Y 483.185,Z 1070.594,A -85,B 0,C 180,E1 19673.211,E2 19673.211} C_VEL
LIN {X 0,Y 486.971,Z 1050.602,A -85,B 0,C 180,E1 19671.679,E2 19671.679} C_VEL
LIN {X 0,Y 490.834,Z 1028.29,A -85,B 0,C 180,E1 19670.235,E2 19670.235} C_VEL
LIN {X 0,Y 494.089,Z 1007.594,A -85,B 0,C 180,E1 19669.107,E2 19669.107} C_VEL
LIN {X 0,Y 497.285,Z 983.886,A -85,B 0,C 180,E1 19668.046,E2 19668.046} C_VEL
LIN {X 0,Y 499.741,Z 962.554,A -85,B 0,C 180,E1 19667.277,E2 19667.277} C_VEL
LIN {X 0,Y 502.018,Z 937.672,A -85,B 0,C 180,E1 19666.592,E2 19666.592} C_VEL
LIN {X 0,Y 503.419,Z 915.54,A -85,B 0,C 180,E1 19666.146,E2 19666.146} C_VEL
LIN {X 0,Y 513.606,Z 671.851,A -85,B 0,C 180,E1 19662.258,E2 19662.258} C_VEL
LIN {X 0,Y 516.062,Z 611.643,A -85,B 0,C 180,E1 19661.298,E2 19661.298} C_VEL
LIN {X 0,Y 503.03,Z 590.912,A -85,B 0,C 180,E1 19659.334,E2 19659.334} C_VEL
LIN {X 0,Y 489.157,Z 570.851,A -85,B 0,C 180,E1 19657.086,E2 19657.086} C_VEL
LIN {X 0,Y 479.666,Z 557.927,A -85,B 0,C 180,E1 19655.409,E2 19655.409} C_VEL
LIN {X 0,Y 473.146,Z 544.537,A -85,B 0,C 180,E1 19652.464,E2 19652.464} C_VEL
LIN {X 0,Y 468.261,Z 535.198,A -85,B 0,C 180,E1 19650.119,E2 19650.119} C_VEL
LIN {X 0,Y 465.771,Z 530.551,A -85,B 0,C 180,E1 19648.856,E2 19648.856} C_VEL
LIN {X 0,Y 463.21,Z 525.755,A -85,B 0,C 180,E1 19647.482,E2 19647.482} C_VEL
LIN {X 0,Y 461.233,Z 522.176,A -85,B 0,C 180,E1 19646.386,E2 19646.386} C_VEL
LIN {X 0,Y 460.341,Z 520.625,A -85,B 0,C 180,E1 19645.886,E2 19645.886} C_VEL
LIN {X 0,Y 458.422,Z 517.268,A -85,B 0,C 180,E1 19644.758,E2 19644.758} C_VEL
LIN {X 0,Y 458.228,Z 516.229,A -85,B 0,C 180,E1 19644.357,E2 19644.357} C_VEL
LIN {X 0,Y 458.194,Z 516.127,A -85,B 0,C 180,E1 19640.837,E2 19640.837} C_VEL
LIN {X 0,Y 458.218,Z 516.123,A -85,B 0,C 180,E1 19637.264,E2 19637.264} C_VEL
LIN {X 0,Y 458.24,Z 516.127,A -85,B 0,C 180,E1 19633.631,E2 19633.631} C_VEL
LIN {X 0,Y 458.218,Z 516.146,A -85,B 0,C 180,E1 19629.927,E2 19629.927} C_VEL
LIN {X 0,Y 458.202,Z 516.146,A -85,B 0,C 180,E1 19626.264,E2 19626.264} C_VEL
LIN {X 0,Y 458.203,Z 516.127,A -85,B 0,C 180,E1 19622.501,E2 19622.501} C_VEL
LIN {X 0,Y 458.235,Z 516.117,A -85,B 0,C 180,E1 19619,E2 19619} C_VEL
LIN {X 0,Y 458.225,Z 516.131,A -85,B 0,C 180,E1 19615.369,E2 19615.369} C_VEL
LIN {X 0,Y 458.209,Z 516.155,A -85,B 0,C 180,E1 19611.719,E2 19611.719} C_VEL
LIN {X 0,Y 458.209,Z 516.142,A -85,B 0,C 180,E1 19608.035,E2 19608.035} C_VEL
LIN {X 0,Y 458.233,Z 516.124,A -85,B 0,C 180,E1 19604.431,E2 19604.431} C_VEL
LIN {X 0,Y 458.235,Z 516.121,A -85,B 0,C 180,E1 19600.762,E2 19600.762} C_VEL
LIN {X 0,Y 458.216,Z 516.125,A -85,B 0,C 180,E1 19597.144,E2 19597.144} C_VEL
LIN {X 0,Y 458.262,Z 516.437,A -85,B 0,C 180,E1 19595,E2 19595} C_VEL
LIN {X 0,Y 459.92,Z 520.147,A -85,B 0,C 180,E1 19593.811,E2 19593.811} C_VEL
LIN {X 0,Y 461.125,Z 521.877,A -85,B 0,C 180,E1 19593.191,E2 19593.191} C_VEL
LIN {X 0,Y 463.269,Z 525.838,A -85,B 0,C 180,E1 19591.973,E2 19591.973} C_VEL
LIN {X 0,Y 466.537,Z 532.128,A -85,B 0,C 180,E1 19590.183,E2 19590.183} C_VEL
LIN {X 0,Y 469.477,Z 537.933,A -85,B 0,C 180,E1 19588.652,E2 19588.652} C_VEL
LIN {X 0,Y 473.273,Z 545.203,A -85,B 0,C 180,E1 19586.825,E2 19586.825} C_VEL
LIN {X 0,Y 479.378,Z 557.983,A -85,B 0,C 180,E1 19583.971,E2 19583.971} C_VEL
LIN {X 0,Y 485.791,Z 572.423,A -85,B 0,C 180,E1 19581.114,E2 19581.114} C_VEL
LIN {X 0,Y 492.449,Z 588.754,A -85,B 0,C 180,E1 19578.242,E2 19578.242} C_VEL
LIN {X 0,Y 498.968,Z 606.458,A -85,B 0,C 180,E1 19575.463,E2 19575.463} C_VEL
LIN {X 0,Y 500.321,Z 610.568,A -85,B 0,C 180,E1 19574.866,E2 19574.866} C_VEL
LIN {X 0,Y 498.068,Z 625.287,A -85,B 0,C 180,E1 19573.617,E2 19573.617} C_VEL
LIN {X 0,Y 505.938,Z 676.469,A -85,B 0,C 180,E1 19571.696,E2 19571.696} C_VEL
LIN {X 0,Y 509.657,Z 703.677,A -85,B 0,C 180,E1 19570.788,E2 19570.788} C_VEL
LIN {X 0,Y 502.045,Z 951.04,A -85,B 0,C 180,E1 19567.292,E2 19567.292} C_VEL
LIN {X 0,Y 500.335,Z 973.387,A -85,B 0,C 180,E1 19566.815,E2 19566.815} C_VEL
LIN {X 0,Y 498.207,Z 993.756,A -85,B 0,C 180,E1 19566.215,E2 19566.215} C_VEL
LIN {X 0,Y 495.393,Z 1014.486,A -85,B 0,C 180,E1 19565.398,E2 19565.398} C_VEL
LIN {X 0,Y 491.942,Z 1035.963,A -85,B 0,C 180,E1 19564.334,E2 19564.334} C_VEL
LIN {X 0,Y 488.329,Z 1055.686,A -85,B 0,C 180,E1 19563.127,E2 19563.127} C_VEL
LIN {X 0,Y 484.441,Z 1074.226,A -85,B 0,C 180,E1 19561.747,E2 19561.747} C_VEL
LIN {X 0,Y 480.431,Z 1092.123,A -85,B 0,C 180,E1 19560.172,E2 19560.172} C_VEL
LIN {X 0,Y 476.467,Z 1108.609,A -85,B 0,C 180,E1 19558.448,E2 19558.448} C_VEL
LIN {X 0,Y 472.456,Z 1124.676,A -85,B 0,C 180,E1 19556.462,E2 19556.462} C_VEL
LIN {X 0,Y 468.724,Z 1139.475,A -85,B 0,C 180,E1 19554.311,E2 19554.311} C_VEL
LIN {X 0,Y 465.469,Z 1152.345,A -85,B 0,C 180,E1 19552.081,E2 19552.081} C_VEL
LIN {X 0,Y 462.519,Z 1164.547,A -85,B 0,C 180,E1 19549.577,E2 19549.577} C_VEL
LIN {X 0,Y 461.698,Z 1168.191,A -85,B 0,C 180,E1 19548.743,E2 19548.743} C_VEL
LIN {X 0,Y 459.97,Z 1171.808,A -85,B 0,C 180,E1 19547.916,E2 19547.916} C_VEL
LIN {X 0,Y 452.022,Z 1180.641,A -85,B 0,C 180,E1 19545.698,E2 19545.698} C_VEL
LIN {X 0,Y 450.781,Z 1183.06,A -85,B 0,C 180,E1 19544.928,E2 19544.928} C_VEL
LIN {X 0,Y 449.46,Z 1190.458,A -85,B 0,C 180,E1 19542.201,E2 19542.201} C_VEL
LIN {X 0,Y 448.62,Z 1196.333,A -85,B 0,C 180,E1 19539.364,E2 19539.364} C_VEL
LIN {X 0,Y 448.165,Z 1200.758,A -85,B 0,C 180,E1 19536.405,E2 19536.405} C_VEL
LIN {X 0,Y 448.006,Z 1203.475,A -85,B 0,C 180,E1 19533.583,E2 19533.583} C_VEL
LIN {X 0,Y 447.966,Z 1204.569,A -85,B 0,C 180,E1 19530.767,E2 19530.767} C_VEL
LIN {X 0,Y 447.976,Z 1204.306,A -85,B 0,C 180,E1 19527.953,E2 19527.953} C_VEL
LIN {X 0,Y 448.048,Z 1202.598,A -85,B 0,C 180,E1 19525.264,E2 19525.264} C_VEL
LIN {X 0,Y 448.308,Z 1199.197,A -85,B 0,C 180,E1 19522.31,E2 19522.31} C_VEL
LIN {X 0,Y 448.846,Z 1194.593,A -85,B 0,C 180,E1 19519.605,E2 19519.605} C_VEL
LIN {X 0,Y 449.851,Z 1188.077,A -85,B 0,C 180,E1 19516.766,E2 19516.766} C_VEL
LIN {X 0,Y 451.399,Z 1180.133,A -85,B 0,C 180,E1 19514.02,E2 19514.02} C_VEL
LIN {X 0,Y 453.53,Z 1170.544,A -85,B 0,C 180,E1 19511.357,E2 19511.357} C_VEL
LIN {X 0,Y 456.242,Z 1159.432,A -85,B 0,C 180,E1 19508.802,E2 19508.802} C_VEL
LIN {X 0,Y 459.53,Z 1146.797,A -85,B 0,C 180,E1 19506.356,E2 19506.356} C_VEL
LIN {X 0,Y 463.138,Z 1133.097,A -85,B 0,C 180,E1 19504.145,E2 19504.145} C_VEL
LIN {X 0,Y 467.277,Z 1117.329,A -85,B 0,C 180,E1 19501.987,E2 19501.987} C_VEL
LIN {X 0,Y 471.458,Z 1101.141,A -85,B 0,C 180,E1 19500.107,E2 19500.107} C_VEL
LIN {X 0,Y 475.585,Z 1083.918,A -85,B 0,C 180,E1 19498.433,E2 19498.433} C_VEL
LIN {X 0,Y 479.939,Z 1064.552,A -85,B 0,C 180,E1 19496.848,E2 19496.848} C_VEL
LIN {X 0,Y 483.776,Z 1045.825,A -85,B 0,C 180,E1 19495.572,E2 19495.572} C_VEL
LIN {X 0,Y 487.225,Z 1026.567,A -85,B 0,C 180,E1 19494.496,E2 19494.496} C_VEL
LIN {X 0,Y 490.344,Z 1006.652,A -85,B 0,C 180,E1 19493.581,E2 19493.581} C_VEL
LIN {X 0,Y 493.014,Z 985.298,A -85,B 0,C 180,E1 19492.827,E2 19492.827} C_VEL
LIN {X 0,Y 495.257,Z 962.152,A -85,B 0,C 180,E1 19492.227,E2 19492.227} C_VEL
LIN {X 0,Y 496.562,Z 939.63,A -85,B 0,C 180,E1 19491.825,E2 19491.825} C_VEL
LIN {X 0,Y 503.906,Z 703.383,A -85,B 0,C 180,E1 19488.459,E2 19488.459} C_VEL
LIN {X 0,Y 496.392,Z 651.176,A -85,B 0,C 180,E1 19486.576,E2 19486.576} C_VEL
LIN {X 0,Y 492.253,Z 623.646,A -85,B 0,C 180,E1 19485.477,E2 19485.477} C_VEL
LIN {X 0,Y 493.793,Z 614.102,A -85,B 0,C 180,E1 19484.64,E2 19484.64} C_VEL
LIN {X 0,Y 487.678,Z 596.828,A -85,B 0,C 180,E1 19481.944,E2 19481.944} C_VEL
LIN {X 0,Y 481.391,Z 580.827,A -85,B 0,C 180,E1 19479.156,E2 19479.156} C_VEL
LIN {X 0,Y 474.741,Z 565.495,A -85,B 0,C 180,E1 19476.138,E2 19476.138} C_VEL
LIN {X 0,Y 469.148,Z 553.681,A -85,B 0,C 180,E1 19473.505,E2 19473.505} C_VEL
LIN {X 0,Y 464.84,Z 544.963,A -85,B 0,C 180,E1 19471.358,E2 19471.358} C_VEL
LIN {X 0,Y 462.416,Z 540.306,A -85,B 0,C 180,E1 19470.11,E2 19470.11} C_VEL
LIN {X 0,Y 460.342,Z 536.185,A -85,B 0,C 180,E1 19468.971,E2 19468.971} C_VEL
LIN {X 0,Y 457.851,Z 531.5,A -85,B 0,C 180,E1 19467.58,E2 19467.58} C_VEL
LIN {X 0,Y 455.255,Z 526.716,A -85,B 0,C 180,E1 19466.057,E2 19466.057} C_VEL
LIN {X 0,Y 453.252,Z 522.875,A -85,B 0,C 180,E1 19464.781,E2 19464.781} C_VEL
LIN {X 0,Y 450.599,Z 518.525,A -85,B 0,C 180,E1 19463.127,E2 19463.127} C_VEL
LIN {X 0,Y 450.28,Z 517.219,A -85,B 0,C 180,E1 19462.592,E2 19462.592} C_VEL
LIN {X 0,Y 450.283,Z 517.109,A -85,B 0,C 180,E1 19458.918,E2 19458.918} C_VEL
LIN {X 0,Y 450.301,Z 517.107,A -85,B 0,C 180,E1 19455.19,E2 19455.19} C_VEL
LIN {X 0,Y 450.285,Z 517.119,A -85,B 0,C 180,E1 19451.528,E2 19451.528} C_VEL
LIN {X 0,Y 450.264,Z 517.145,A -85,B 0,C 180,E1 19447.914,E2 19447.914} C_VEL
LIN {X 0,Y 450.265,Z 517.13,A -85,B 0,C 180,E1 19444.203,E2 19444.203} C_VEL
LIN {X 0,Y 450.292,Z 517.109,A -85,B 0,C 180,E1 19440.509,E2 19440.509} C_VEL
LIN {X 0,Y 450.292,Z 517.106,A -85,B 0,C 180,E1 19436.818,E2 19436.818} C_VEL
LIN {X 0,Y 450.274,Z 517.12,A -85,B 0,C 180,E1 19433.113,E2 19433.113} C_VEL
LIN {X 0,Y 450.26,Z 517.143,A -85,B 0,C 180,E1 19429.379,E2 19429.379} C_VEL
LIN {X 0,Y 450.257,Z 517.138,A -85,B 0,C 180,E1 19425.598,E2 19425.598} C_VEL
LIN {X 0,Y 450.287,Z 517.118,A -85,B 0,C 180,E1 19422.022,E2 19422.022} C_VEL
LIN {X 0,Y 450.303,Z 517.119,A -85,B 0,C 180,E1 19418.234,E2 19418.234} C_VEL
LIN {X 0,Y 450.358,Z 517.697,A -85,B 0,C 180,E1 19417.55,E2 19417.55} C_VEL
LIN {X 0,Y 452.013,Z 521.166,A -85,B 0,C 180,E1 19416.315,E2 19416.315} C_VEL
LIN {X 0,Y 453.26,Z 522.834,A -85,B 0,C 180,E1 19415.637,E2 19415.637} C_VEL
LIN {X 0,Y 455.02,Z 526.401,A -85,B 0,C 180,E1 19414.488,E2 19414.488} C_VEL
LIN {X 0,Y 456.178,Z 528.208,A -85,B 0,C 180,E1 19413.86,E2 19413.86} C_VEL
LIN {X 0,Y 458.17,Z 531.882,A -85,B 0,C 180,E1 19412.723,E2 19412.723} C_VEL
LIN {X 0,Y 461.762,Z 538.714,A -85,B 0,C 180,E1 19410.764,E2 19410.764} C_VEL
LIN {X 0,Y 466.114,Z 546.958,A -85,B 0,C 180,E1 19408.582,E2 19408.582} C_VEL
LIN {X 0,Y 472.348,Z 559.437,A -85,B 0,C 180,E1 19405.694,E2 19405.694} C_VEL
LIN {X 0,Y 483.973,Z 575.174,A -85,B 0,C 180,E1 19403.56,E2 19403.56} C_VEL
LIN {X 0,Y 496.841,Z 593.705,A -85,B 0,C 180,E1 19401.4,E2 19401.4} C_VEL
LIN {X 0,Y 509.694,Z 614.008,A -85,B 0,C 180,E1 19399.393,E2 19399.393} C_VEL
LIN {X 0,Y 510.48,Z 615.79,A -85,B 0,C 180,E1 19399.265,E2 19399.265} C_VEL
LIN {X 0,Y 500.041,Z 854.249,A -85,B 0,C 180,E1 19395.458,E2 19395.458} C_VEL
LIN {X 0,Y 496.839,Z 926.092,A -85,B 0,C 180,E1 19394.274,E2 19394.274} C_VEL
LIN {X 0,Y 494.825,Z 950.562,A -85,B 0,C 180,E1 19393.688,E2 19393.688} C_VEL
LIN {X 0,Y 492.376,Z 973.951,A -85,B 0,C 180,E1 19392.945,E2 19392.945} C_VEL
LIN {X 0,Y 489.38,Z 996.682,A -85,B 0,C 180,E1 19392.007,E2 19392.007} C_VEL
LIN {X 0,Y 485.965,Z 1019.493,A -85,B 0,C 180,E1 19390.865,E2 19390.865} C_VEL
LIN {X 0,Y 482.303,Z 1040.544,A -85,B 0,C 180,E1 19389.579,E2 19389.579} C_VEL
LIN {X 0,Y 478.345,Z 1061.718,A -85,B 0,C 180,E1 19388.07,E2 19388.07} C_VEL
LIN {X 0,Y 474.134,Z 1082.111,A -85,B 0,C 180,E1 19386.34,E2 19386.34} C_VEL
LIN {X 0,Y 470.051,Z 1101.336,A -85,B 0,C 180,E1 19384.459,E2 19384.459} C_VEL
LIN {X 0,Y 466.117,Z 1119.042,A -85,B 0,C 180,E1 19382.43,E2 19382.43} C_VEL
LIN {X 0,Y 462.47,Z 1135.742,A -85,B 0,C 180,E1 19380.248,E2 19380.248} C_VEL
LIN {X 0,Y 458.93,Z 1151.762,A -85,B 0,C 180,E1 19377.801,E2 19377.801} C_VEL
LIN {X 0,Y 455.846,Z 1166.649,A -85,B 0,C 180,E1 19375.184,E2 19375.184} C_VEL
LIN {X 0,Y 453.377,Z 1179.345,A -85,B 0,C 180,E1 19372.565,E2 19372.565} C_VEL
LIN {X 0,Y 451.288,Z 1191.407,A -85,B 0,C 180,E1 19369.669,E2 19369.669} C_VEL
LIN {X 0,Y 449.928,Z 1200.535,A -85,B 0,C 180,E1 19367.058,E2 19367.058} C_VEL
LIN {X 0,Y 448.921,Z 1209.056,A -85,B 0,C 180,E1 19364.182,E2 19364.182} C_VEL
LIN {X 0,Y 448.322,Z 1215.731,A -85,B 0,C 180,E1 19361.318,E2 19361.318} C_VEL
LIN {X 0,Y 448.062,Z 1220.643,A -85,B 0,C 180,E1 19358.66,E2 19358.66} C_VEL
LIN {X 0,Y 447.934,Z 1224.612,A -85,B 0,C 180,E1 19355.636,E2 19355.636} C_VEL
LIN {X 0,Y 447.923,Z 1226.566,A -85,B 0,C 180,E1 19353.199,E2 19353.199} C_VEL
LIN {X 0,Y 447.925,Z 1227.458,A -85,B 0,C 180,E1 19350.767,E2 19350.767} C_VEL
LIN {X 0,Y 447.937,Z 1227.206,A -85,B 0,C 180,E1 19347.953,E2 19347.953} C_VEL
LIN {X 0,Y 447.927,Z 1225.33,A -85,B 0,C 180,E1 19345.134,E2 19345.134} C_VEL
LIN {X 0,Y 447.976,Z 1222.596,A -85,B 0,C 180,E1 19342.691,E2 19342.691} C_VEL
LIN {X 0,Y 448.172,Z 1218.118,A -85,B 0,C 180,E1 19339.849,E2 19339.849} C_VEL
LIN {X 0,Y 448.656,Z 1211.66,A -85,B 0,C 180,E1 19336.886,E2 19336.886} C_VEL
LIN {X 0,Y 449.461,Z 1204.227,A -85,B 0,C 180,E1 19334.12,E2 19334.12} C_VEL
LIN {X 0,Y 450.759,Z 1194.712,A -85,B 0,C 180,E1 19331.238,E2 19331.238} C_VEL
LIN {X 0,Y 452.434,Z 1184.494,A -85,B 0,C 180,E1 19328.614,E2 19328.614} C_VEL
LIN {X 0,Y 454.904,Z 1171.244,A -85,B 0,C 180,E1 19325.731,E2 19325.731} C_VEL
LIN {X 0,Y 457.456,Z 1158.701,A -85,B 0,C 180,E1 19323.378,E2 19323.378} C_VEL
LIN {X 0,Y 460.883,Z 1142.689,A -85,B 0,C 180,E1 19320.783,E2 19320.783} C_VEL
LIN {X 0,Y 464.257,Z 1127.356,A -85,B 0,C 180,E1 19318.628,E2 19318.628} C_VEL
LIN {X 0,Y 468.399,Z 1108.667,A -85,B 0,C 180,E1 19316.36,E2 19316.36} C_VEL
LIN {X 0,Y 472.17,Z 1091.296,A -85,B 0,C 180,E1 19314.534,E2 19314.534} C_VEL
LIN {X 0,Y 476.457,Z 1070.632,A -85,B 0,C 180,E1 19312.665,E2 19312.665} C_VEL
LIN {X 0,Y 480.193,Z 1051.637,A -85,B 0,C 180,E1 19311.19,E2 19311.19} C_VEL
LIN {X 0,Y 484.188,Z 1029.553,A -85,B 0,C 180,E1 19309.733,E2 19309.733} C_VEL
LIN {X 0,Y 487.467,Z 1009.446,A -85,B 0,C 180,E1 19308.617,E2 19308.617} C_VEL
LIN {X 0,Y 490.901,Z 985.201,A -85,B 0,C 180,E1 19307.506,E2 19307.506} C_VEL
LIN {X 0,Y 493.415,Z 964.103,A -85,B 0,C 180,E1 19306.731,E2 19306.731} C_VEL
LIN {X 0,Y 495.856,Z 938.69,A -85,B 0,C 180,E1 19306.015,E2 19306.015} C_VEL
LIN {X 0,Y 497.309,Z 916.666,A -85,B 0,C 180,E1 19305.564,E2 19305.564} C_VEL
LIN {X 0,Y 507.813,Z 673.93,A -85,B 0,C 180,E1 19301.658,E2 19301.658} C_VEL
LIN {X 0,Y 510.293,Z 615.059,A -85,B 0,C 180,E1 19300.712,E2 19300.712} C_VEL
LIN {X 0,Y 497.781,Z 595.217,A -85,B 0,C 180,E1 19298.771,E2 19298.771} C_VEL
LIN {X 0,Y 484.86,Z 576.441,A -85,B 0,C 180,E1 19296.62,E2 19296.62} C_VEL
LIN {X 0,Y 474.87,Z 562.924,A -85,B 0,C 180,E1 19294.83,E2 19294.83} C_VEL
LIN {X 0,Y 472.138,Z 559.116,A -85,B 0,C 180,E1 19294.287,E2 19294.287} C_VEL
LIN {X 0,Y 466.994,Z 548.955,A -85,B 0,C 180,E1 19291.928,E2 19291.928} C_VEL
LIN {X 0,Y 463.294,Z 541.455,A -85,B 0,C 180,E1 19290.047,E2 19290.047} C_VEL
LIN {X 0,Y 460.327,Z 536.115,A -85,B 0,C 180,E1 19288.546,E2 19288.546} C_VEL
LIN {X 0,Y 458.058,Z 531.744,A -85,B 0,C 180,E1 19287.285,E2 19287.285} C_VEL
LIN {X 0,Y 456.103,Z 528.004,A -85,B 0,C 180,E1 19286.145,E2 19286.145} C_VEL
LIN {X 0,Y 453.48,Z 523.543,A -85,B 0,C 180,E1 19284.629,E2 19284.629} C_VEL
LIN {X 0,Y 452.732,Z 521.962,A -85,B 0,C 180,E1 19284.116,E2 19284.116} C_VEL
LIN {X 0,Y 450.613,Z 518.701,A -85,B 0,C 180,E1 19282.85,E2 19282.85} C_VEL
LIN {X 0,Y 450.296,Z 517.286,A -85,B 0,C 180,E1 19282.316,E2 19282.316} C_VEL
LIN {X 0,Y 450.26,Z 517.139,A -85,B 0,C 180,E1 19278.65,E2 19278.65} C_VEL
LIN {X 0,Y 450.267,Z 517.144,A -85,B 0,C 180,E1 19274.928,E2 19274.928} C_VEL
LIN {X 0,Y 450.289,Z 517.121,A -85,B 0,C 180,E1 19271.269,E2 19271.269} C_VEL
LIN {X 0,Y 450.3,Z 517.104,A -85,B 0,C 180,E1 19267.528,E2 19267.528} C_VEL
LIN {X 0,Y 450.272,Z 517.106,A -85,B 0,C 180,E1 19263.82,E2 19263.82} C_VEL
LIN {X 0,Y 450.26,Z 517.123,A -85,B 0,C 180,E1 19260.127,E2 19260.127} C_VEL
LIN {X 0,Y 450.275,Z 517.144,A -85,B 0,C 180,E1 19256.435,E2 19256.435} C_VEL
LIN {X 0,Y 450.302,Z 517.122,A -85,B 0,C 180,E1 19252.729,E2 19252.729} C_VEL
LIN {X 0,Y 450.295,Z 517.109,A -85,B 0,C 180,E1 19248.943,E2 19248.943} C_VEL
LIN {X 0,Y 450.285,Z 517.108,A -85,B 0,C 180,E1 19245.205,E2 19245.205} C_VEL
LIN {X 0,Y 450.269,Z 517.114,A -85,B 0,C 180,E1 19241.485,E2 19241.485} C_VEL
LIN {X 0,Y 450.271,Z 517.118,A -85,B 0,C 180,E1 19237.683,E2 19237.683} C_VEL
LIN {X 0,Y 450.366,Z 517.628,A -85,B 0,C 180,E1 19236.999,E2 19236.999} C_VEL
LIN {X 0,Y 452.202,Z 521.421,A -85,B 0,C 180,E1 19235.639,E2 19235.639} C_VEL
LIN {X 0,Y 453.274,Z 522.928,A -85,B 0,C 180,E1 19235.04,E2 19235.04} C_VEL
LIN {X 0,Y 455.223,Z 526.678,A -85,B 0,C 180,E1 19233.801,E2 19233.801} C_VEL
LIN {X 0,Y 456.286,Z 528.654,A -85,B 0,C 180,E1 19233.165,E2 19233.165} C_VEL
LIN {X 0,Y 458.889,Z 533.504,A -85,B 0,C 180,E1 19231.674,E2 19231.674} C_VEL
LIN {X 0,Y 461.308,Z 538.032,A -85,B 0,C 180,E1 19230.359,E2 19230.359} C_VEL
LIN {X 0,Y 465.938,Z 547.101,A -85,B 0,C 180,E1 19227.955,E2 19227.955} C_VEL
LIN {X 0,Y 471.814,Z 559.199,A -85,B 0,C 180,E1 19225.096,E2 19225.096} C_VEL
LIN {X 0,Y 478.345,Z 573.703,A -85,B 0,C 180,E1 19222.08,E2 19222.08} C_VEL
LIN {X 0,Y 484.856,Z 589.52,A -85,B 0,C 180,E1 19219.176,E2 19219.176} C_VEL
LIN {X 0,Y 491.244,Z 606.698,A -85,B 0,C 180,E1 19216.369,E2 19216.369} C_VEL
LIN {X 0,Y 493.708,Z 614.449,A -85,B 0,C 180,E1 19215.221,E2 19215.221} C_VEL
LIN {X 0,Y 492.196,Z 624.568,A -85,B 0,C 180,E1 19214.37,E2 19214.37} C_VEL
LIN {X 0,Y 499.91,Z 675.577,A -85,B 0,C 180,E1 19212.413,E2 19212.413} C_VEL
LIN {X 0,Y 503.902,Z 704.978,A -85,B 0,C 180,E1 19211.405,E2 19211.405} C_VEL
LIN {X 0,Y 495.984,Z 950.817,A -85,B 0,C 180,E1 19207.895,E2 19207.895} C_VEL
LIN {X 0,Y 494.213,Z 973.238,A -85,B 0,C 180,E1 19207.413,E2 19207.413} C_VEL
LIN {X 0,Y 491.953,Z 994.052,A -85,B 0,C 180,E1 19206.793,E2 19206.793} C_VEL
LIN {X 0,Y 489.135,Z 1014.187,A -85,B 0,C 180,E1 19205.993,E2 19205.993} C_VEL
LIN {X 0,Y 485.565,Z 1035.705,A -85,B 0,C 180,E1 19204.921,E2 19204.921} C_VEL
LIN {X 0,Y 482.022,Z 1054.398,A -85,B 0,C 180,E1 19203.773,E2 19203.773} C_VEL
LIN {X 0,Y 477.988,Z 1073.216,A -85,B 0,C 180,E1 19202.378,E2 19202.378} C_VEL
LIN {X 0,Y 473.933,Z 1090.856,A -85,B 0,C 180,E1 19200.831,E2 19200.831} C_VEL
LIN {X 0,Y 469.662,Z 1107.929,A -85,B 0,C 180,E1 19199.038,E2 19199.038} C_VEL
LIN {X 0,Y 465.341,Z 1124.624,A -85,B 0,C 180,E1 19196.96,E2 19196.96} C_VEL
LIN {X 0,Y 461.443,Z 1139.458,A -85,B 0,C 180,E1 19194.78,E2 19194.78} C_VEL
LIN {X 0,Y 457.967,Z 1152.635,A -85,B 0,C 180,E1 19192.462,E2 19192.462} C_VEL
LIN {X 0,Y 454.882,Z 1164.81,A -85,B 0,C 180,E1 19189.919,E2 19189.919} C_VEL
LIN {X 0,Y 452.449,Z 1175.263,A -85,B 0,C 180,E1 19187.311,E2 19187.311} C_VEL
LIN {X 0,Y 450.781,Z 1183.06,A -85,B 0,C 180,E1 19184.928,E2 19184.928} C_VEL
LIN {X 0,Y 449.278,Z 1185.873,A -85,B 0,C 180,E1 19184.023,E2 19184.023} C_VEL
LIN {X 0,Y 441.997,Z 1192.504,A -85,B 0,C 180,E1 19181.601,E2 19181.601} C_VEL
LIN {X 0,Y 440.991,Z 1194.266,A -85,B 0,C 180,E1 19180.776,E2 19180.776} C_VEL
LIN {X 0,Y 440.366,Z 1199.065,A -85,B 0,C 180,E1 19177.961,E2 19177.961} C_VEL
LIN {X 0,Y 440.065,Z 1202.615,A -85,B 0,C 180,E1 19174.953,E2 19174.953} C_VEL
LIN {X 0,Y 439.982,Z 1204.398,A -85,B 0,C 180,E1 19172.214,E2 19172.214} C_VEL
LIN {X 0,Y 439.965,Z 1204.79,A -85,B 0,C 180,E1 19169.219,E2 19169.219} C_VEL
LIN {X 0,Y 440.01,Z 1203.747,A -85,B 0,C 180,E1 19166.352,E2 19166.352} C_VEL
LIN {X 0,Y 440.18,Z 1201.083,A -85,B 0,C 180,E1 19163.479,E2 19163.479} C_VEL
LIN {X 0,Y 440.647,Z 1196.732,A -85,B 0,C 180,E1 19160.466,E2 19160.466} C_VEL
LIN {X 0,Y 441.522,Z 1190.898,A -85,B 0,C 180,E1 19157.577,E2 19157.577} C_VEL
LIN {X 0,Y 442.894,Z 1183.638,A -85,B 0,C 180,E1 19154.819,E2 19154.819} C_VEL
LIN {X 0,Y 444.896,Z 1174.736,A -85,B 0,C 180,E1 19152.068,E2 19152.068} C_VEL
LIN {X 0,Y 447.508,Z 1164.206,A -85,B 0,C 180,E1 19149.423,E2 19149.423} C_VEL
LIN {X 0,Y 450.735,Z 1152.069,A -85,B 0,C 180,E1 19146.881,E2 19146.881} C_VEL
LIN {X 0,Y 454.314,Z 1139.133,A -85,B 0,C 180,E1 19144.586,E2 19144.586} C_VEL
LIN {X 0,Y 458.254,Z 1124.725,A -85,B 0,C 180,E1 19142.448,E2 19142.448} C_VEL
LIN {X 0,Y 462.75,Z 1108.03,A -85,B 0,C 180,E1 19140.344,E2 19140.344} C_VEL
LIN {X 0,Y 467.048,Z 1091.472,A -85,B 0,C 180,E1 19138.582,E2 19138.582} C_VEL
LIN {X 0,Y 471.22,Z 1074.061,A -85,B 0,C 180,E1 19137.026,E2 19137.026} C_VEL
LIN {X 0,Y 475.385,Z 1055.434,A -85,B 0,C 180,E1 19135.617,E2 19135.617} C_VEL
LIN {X 0,Y 479.223,Z 1035.869,A -85,B 0,C 180,E1 19134.401,E2 19134.401} C_VEL
LIN {X 0,Y 482.91,Z 1014.433,A -85,B 0,C 180,E1 19133.321,E2 19133.321} C_VEL
LIN {X 0,Y 485.831,Z 994.239,A -85,B 0,C 180,E1 19132.511,E2 19132.511} C_VEL
LIN {X 0,Y 488.238,Z 972.862,A -85,B 0,C 180,E1 19131.868,E2 19131.868} C_VEL
LIN {X 0,Y 490.062,Z 950.365,A -85,B 0,C 180,E1 19131.383,E2 19131.383} C_VEL
LIN {X 0,Y 498.24,Z 705.005,A -85,B 0,C 180,E1 19127.836,E2 19127.836} C_VEL
LIN {X 0,Y 490.924,Z 653.064,A -85,B 0,C 180,E1 19125.928,E2 19125.928} C_VEL
LIN {X 0,Y 486.448,Z 622.857,A -85,B 0,C 180,E1 19124.704,E2 19124.704} C_VEL
LIN {X 0,Y 487.244,Z 617.683,A -85,B 0,C 180,E1 19124.245,E2 19124.245} C_VEL
LIN {X 0,Y 481.216,Z 600.568,A -85,B 0,C 180,E1 19121.516,E2 19121.516} C_VEL
LIN {X 0,Y 475.299,Z 585.425,A -85,B 0,C 180,E1 19118.822,E2 19118.822} C_VEL
LIN {X 0,Y 469.037,Z 570.751,A -85,B 0,C 180,E1 19115.891,E2 19115.891} C_VEL
LIN {X 0,Y 463.378,Z 558.69,A -85,B 0,C 180,E1 19113.154,E2 19113.154} C_VEL
LIN {X 0,Y 459.296,Z 550.355,A -85,B 0,C 180,E1 19111.061,E2 19111.061} C_VEL
LIN {X 0,Y 457.142,Z 546.122,A -85,B 0,C 180,E1 19109.914,E2 19109.914} C_VEL
LIN {X 0,Y 455.078,Z 542.022,A -85,B 0,C 180,E1 19108.76,E2 19108.76} C_VEL
LIN {X 0,Y 452.625,Z 537.367,A -85,B 0,C 180,E1 19107.354,E2 19107.354} C_VEL
LIN {X 0,Y 450.303,Z 532.932,A -85,B 0,C 180,E1 19105.939,E2 19105.939} C_VEL
LIN {X 0,Y 447.677,Z 528.107,A -85,B 0,C 180,E1 19104.266,E2 19104.266} C_VEL
LIN {X 0,Y 445.552,Z 524.357,A -85,B 0,C 180,E1 19102.845,E2 19102.845} C_VEL
LIN {X 0,Y 444.603,Z 522.774,A -85,B 0,C 180,E1 19102.199,E2 19102.199} C_VEL
LIN {X 0,Y 442.52,Z 519.117,A -85,B 0,C 180,E1 19100.64,E2 19100.64} C_VEL
LIN {X 0,Y 442.345,Z 518.204,A -85,B 0,C 180,E1 19100.096,E2 19100.096} C_VEL
LIN {X 0,Y 442.327,Z 518.121,A -85,B 0,C 180,E1 19096.413,E2 19096.413} C_VEL
LIN {X 0,Y 442.349,Z 518.128,A -85,B 0,C 180,E1 19092.798,E2 19092.798} C_VEL
LIN {X 0,Y 442.359,Z 518.108,A -85,B 0,C 180,E1 19088.973,E2 19088.973} C_VEL
LIN {X 0,Y 442.344,Z 518.096,A -85,B 0,C 180,E1 19085.318,E2 19085.318} C_VEL
LIN {X 0,Y 442.321,Z 518.1,A -85,B 0,C 180,E1 19081.684,E2 19081.684} C_VEL
LIN {X 0,Y 442.321,Z 518.115,A -85,B 0,C 180,E1 19077.927,E2 19077.927} C_VEL
LIN {X 0,Y 442.34,Z 518.132,A -85,B 0,C 180,E1 19074.162,E2 19074.162} C_VEL
LIN {X 0,Y 442.357,Z 518.109,A -85,B 0,C 180,E1 19070.502,E2 19070.502} C_VEL
LIN {X 0,Y 442.351,Z 518.099,A -85,B 0,C 180,E1 19066.67,E2 19066.67} C_VEL
LIN {X 0,Y 442.319,Z 518.1,A -85,B 0,C 180,E1 19063.045,E2 19063.045} C_VEL
LIN {X 0,Y 442.4,Z 518.437,A -85,B 0,C 180,E1 19059.993,E2 19059.993} C_VEL
LIN {X 0,Y 443.936,Z 521.99,A -85,B 0,C 180,E1 19058.6,E2 19058.6} C_VEL
LIN {X 0,Y 445.415,Z 523.927,A -85,B 0,C 180,E1 19057.705,E2 19057.705} C_VEL
LIN {X 0,Y 447.23,Z 527.536,A -85,B 0,C 180,E1 19056.409,E2 19056.409} C_VEL
LIN {X 0,Y 448.344,Z 529.134,A -85,B 0,C 180,E1 19055.773,E2 19055.773} C_VEL
LIN {X 0,Y 450.369,Z 532.956,A -85,B 0,C 180,E1 19054.487,E2 19054.487} C_VEL
LIN {X 0,Y 451.395,Z 535.003,A -85,B 0,C 180,E1 19053.844,E2 19053.844} C_VEL
LIN {X 0,Y 453.88,Z 539.451,A -85,B 0,C 180,E1 19052.443,E2 19052.443} C_VEL
LIN {X 0,Y 456.862,Z 545.249,A -85,B 0,C 180,E1 19050.787,E2 19050.787} C_VEL
LIN {X 0,Y 461.049,Z 553.354,A -85,B 0,C 180,E1 19048.634,E2 19048.634} C_VEL
LIN {X 0,Y 464.923,Z 560.884,A -85,B 0,C 180,E1 19046.852,E2 19046.852} C_VEL
LIN {X 0,Y 477.514,Z 577.648,A -85,B 0,C 180,E1 19044.437,E2 19044.437} C_VEL
LIN {X 0,Y 489.508,Z 594.83,A -85,B 0,C 180,E1 19042.337,E2 19042.337} C_VEL
LIN {X 0,Y 501.391,Z 613.327,A -85,B 0,C 180,E1 19040.401,E2 19040.401} C_VEL
LIN {X 0,Y 504.779,Z 619.092,A -85,B 0,C 180,E1 19039.867,E2 19039.867} C_VEL
LIN {X 0,Y 494.024,Z 856.989,A -85,B 0,C 180,E1 19036.039,E2 19036.039} C_VEL
LIN {X 0,Y 490.805,Z 926.661,A -85,B 0,C 180,E1 19034.88,E2 19034.88} C_VEL
LIN {X 0,Y 488.717,Z 951.152,A -85,B 0,C 180,E1 19034.286,E2 19034.286} C_VEL
LIN {X 0,Y 486.211,Z 974.308,A -85,B 0,C 180,E1 19033.543,E2 19033.543} C_VEL
LIN {X 0,Y 483.101,Z 997.116,A -85,B 0,C 180,E1 19032.592,E2 19032.592} C_VEL
LIN {X 0,Y 479.59,Z 1019.764,A -85,B 0,C 180,E1 19031.447,E2 19031.447} C_VEL
LIN {X 0,Y 475.854,Z 1040.486,A -85,B 0,C 180,E1 19030.17,E2 19030.17} C_VEL
LIN {X 0,Y 471.865,Z 1061.116,A -85,B 0,C 180,E1 19028.689,E2 19028.689} C_VEL
LIN {X 0,Y 467.492,Z 1081.608,A -85,B 0,C 180,E1 19026.941,E2 19026.941} C_VEL
LIN {X 0,Y 463.232,Z 1100.906,A -85,B 0,C 180,E1 19025.04,E2 19025.04} C_VEL
LIN {X 0,Y 458.999,Z 1119.164,A -85,B 0,C 180,E1 19022.922,E2 19022.922} C_VEL
LIN {X 0,Y 455.09,Z 1136.266,A -85,B 0,C 180,E1 19020.645,E2 19020.645} C_VEL
LIN {X 0,Y 451.571,Z 1151.49,A -85,B 0,C 180,E1 19018.283,E2 19018.283} C_VEL
LIN {X 0,Y 448.343,Z 1166.351,A -85,B 0,C 180,E1 19015.635,E2 19015.635} C_VEL
LIN {X 0,Y 445.842,Z 1178.461,A -85,B 0,C 180,E1 19013.108,E2 19013.108} C_VEL
LIN {X 0,Y 443.699,Z 1190.144,A -85,B 0,C 180,E1 19010.306,E2 19010.306} C_VEL
LIN {X 0,Y 442.07,Z 1200.284,A -85,B 0,C 180,E1 19007.371,E2 19007.371} C_VEL
LIN {X 0,Y 440.993,Z 1208.818,A -85,B 0,C 180,E1 19004.442,E2 19004.442} C_VEL
LIN {X 0,Y 440.35,Z 1215.506,A -85,B 0,C 180,E1 19001.526,E2 19001.526} C_VEL
LIN {X 0,Y 440.068,Z 1220.31,A -85,B 0,C 180,E1 18998.888,E2 18998.888} C_VEL
LIN {X 0,Y 439.94,Z 1224.403,A -85,B 0,C 180,E1 18995.739,E2 18995.739} C_VEL
LIN {X 0,Y 439.928,Z 1226.36,A -85,B 0,C 180,E1 18993.257,E2 18993.257} C_VEL
LIN {X 0,Y 439.928,Z 1227.253,A -85,B 0,C 180,E1 18990.781,E2 18990.781} C_VEL
LIN {X 0,Y 439.939,Z 1227.001,A -85,B 0,C 180,E1 18987.916,E2 18987.916} C_VEL
LIN {X 0,Y 439.926,Z 1225.121,A -85,B 0,C 180,E1 18985.045,E2 18985.045} C_VEL
LIN {X 0,Y 439.975,Z 1222.381,A -85,B 0,C 180,E1 18982.557,E2 18982.557} C_VEL
LIN {X 0,Y 440.199,Z 1217.761,A -85,B 0,C 180,E1 18979.591,E2 18979.591} C_VEL
LIN {X 0,Y 440.72,Z 1211.365,A -85,B 0,C 180,E1 18976.62,E2 18976.62} C_VEL
LIN {X 0,Y 441.626,Z 1203.612,A -85,B 0,C 180,E1 18973.696,E2 18973.696} C_VEL
LIN {X 0,Y 443.037,Z 1193.968,A -85,B 0,C 180,E1 18970.762,E2 18970.762} C_VEL
LIN {X 0,Y 444.952,Z 1183.143,A -85,B 0,C 180,E1 18967.959,E2 18967.959} C_VEL
LIN {X 0,Y 447.475,Z 1170.279,A -85,B 0,C 180,E1 18965.161,E2 18965.161} C_VEL
LIN {X 0,Y 450.547,Z 1156.211,A -85,B 0,C 180,E1 18962.51,E2 18962.51} C_VEL
LIN {X 0,Y 454.025,Z 1140.58,A -85,B 0,C 180,E1 18960.007,E2 18960.007} C_VEL
LIN {X 0,Y 457.952,Z 1123.796,A -85,B 0,C 180,E1 18957.662,E2 18957.662} C_VEL
LIN {X 0,Y 461.98,Z 1106.11,A -85,B 0,C 180,E1 18955.551,E2 18955.551} C_VEL
LIN {X 0,Y 466.302,Z 1086.971,A -85,B 0,C 180,E1 18953.562,E2 18953.562} C_VEL
LIN {X 0,Y 470.393,Z 1067.73,A -85,B 0,C 180,E1 18951.859,E2 18951.859} C_VEL
LIN {X 0,Y 474.684,Z 1046.62,A -85,B 0,C 180,E1 18950.251,E2 18950.251} C_VEL
LIN {X 0,Y 478.297,Z 1026.74,A -85,B 0,C 180,E1 18948.974,E2 18948.974} C_VEL
LIN {X 0,Y 481.983,Z 1004.66,A -85,B 0,C 180,E1 18947.769,E2 18947.769} C_VEL
LIN {X 0,Y 485.116,Z 982.274,A -85,B 0,C 180,E1 18946.781,E2 18946.781} C_VEL
LIN {X 0,Y 487.919,Z 959.218,A -85,B 0,C 180,E1 18945.957,E2 18945.957} C_VEL
LIN {X 0,Y 490.069,Z 935.566,A -85,B 0,C 180,E1 18945.328,E2 18945.328} C_VEL
LIN {X 0,Y 491.634,Z 910.756,A -85,B 0,C 180,E1 18944.843,E2 18944.843} C_VEL
LIN {X 0,Y 502.517,Z 666.382,A -85,B 0,C 180,E1 18940.891,E2 18940.891} C_VEL
LIN {X 0,Y 504.597,Z 618.569,A -85,B 0,C 180,E1 18940.116,E2 18940.116} C_VEL
LIN {X 0,Y 491.728,Z 598.112,A -85,B 0,C 180,E1 18938.053,E2 18938.053} C_VEL
LIN {X 0,Y 478.384,Z 578.823,A -85,B 0,C 180,E1 18935.746,E2 18935.746} C_VEL
LIN {X 0,Y 467.24,Z 564.101,A -85,B 0,C 180,E1 18933.66,E2 18933.66} C_VEL
LIN {X 0,Y 464.365,Z 559.968,A -85,B 0,C 180,E1 18933.009,E2 18933.009} C_VEL
LIN {X 0,Y 459.704,Z 550.756,A -85,B 0,C 180,E1 18930.74,E2 18930.74} C_VEL
LIN {X 0,Y 455.645,Z 542.746,A -85,B 0,C 180,E1 18928.58,E2 18928.58} C_VEL
LIN {X 0,Y 452.857,Z 537.649,A -85,B 0,C 180,E1 18927.055,E2 18927.055} C_VEL
LIN {X 0,Y 450.512,Z 533.121,A -85,B 0,C 180,E1 18925.645,E2 18925.645} C_VEL
LIN {X 0,Y 448.408,Z 529.371,A -85,B 0,C 180,E1 18924.364,E2 18924.364} C_VEL
LIN {X 0,Y 446.878,Z 527.078,A -85,B 0,C 180,E1 18923.471,E2 18923.471} C_VEL
LIN {X 0,Y 444.922,Z 523.098,A -85,B 0,C 180,E1 18922.043,E2 18922.043} C_VEL
LIN {X 0,Y 442.765,Z 519.921,A -85,B 0,C 180,E1 18920.628,E2 18920.628} C_VEL
LIN {X 0,Y 442.37,Z 518.215,A -85,B 0,C 180,E1 18919.906,E2 18919.906} C_VEL
LIN {X 0,Y 442.337,Z 518.104,A -85,B 0,C 180,E1 18916.123,E2 18916.123} C_VEL
LIN {X 0,Y 442.32,Z 518.099,A -85,B 0,C 180,E1 18912.438,E2 18912.438} C_VEL
LIN {X 0,Y 442.322,Z 518.098,A -85,B 0,C 180,E1 18908.711,E2 18908.711} C_VEL
LIN {X 0,Y 442.35,Z 518.111,A -85,B 0,C 180,E1 18905.058,E2 18905.058} C_VEL
LIN {X 0,Y 442.362,Z 518.127,A -85,B 0,C 180,E1 18901.295,E2 18901.295} C_VEL
LIN {X 0,Y 442.342,Z 518.108,A -85,B 0,C 180,E1 18897.538,E2 18897.538} C_VEL
LIN {X 0,Y 442.329,Z 518.098,A -85,B 0,C 180,E1 18893.771,E2 18893.771} C_VEL
LIN {X 0,Y 442.326,Z 518.098,A -85,B 0,C 180,E1 18889.976,E2 18889.976} C_VEL
LIN {X 0,Y 442.346,Z 518.106,A -85,B 0,C 180,E1 18886.27,E2 18886.27} C_VEL
LIN {X 0,Y 442.359,Z 518.117,A -85,B 0,C 180,E1 18882.505,E2 18882.505} C_VEL
LIN {X 0,Y 442.365,Z 518.354,A -85,B 0,C 180,E1 18879.491,E2 18879.491} C_VEL
LIN {X 0,Y 444.099,Z 522.197,A -85,B 0,C 180,E1 18877.914,E2 18877.914} C_VEL
LIN {X 0,Y 445.387,Z 523.83,A -85,B 0,C 180,E1 18877.146,E2 18877.146} C_VEL
LIN {X 0,Y 447.388,Z 527.781,A -85,B 0,C 180,E1 18875.718,E2 18875.718} C_VEL
LIN {X 0,Y 448.423,Z 529.517,A -85,B 0,C 180,E1 18875.075,E2 18875.075} C_VEL
LIN {X 0,Y 451.117,Z 534.465,A -85,B 0,C 180,E1 18873.402,E2 18873.402} C_VEL
LIN {X 0,Y 453.81,Z 539.657,A -85,B 0,C 180,E1 18871.799,E2 18871.799} C_VEL
LIN {X 0,Y 456.216,Z 544.271,A -85,B 0,C 180,E1 18870.453,E2 18870.453} C_VEL
LIN {X 0,Y 460.341,Z 552.232,A -85,B 0,C 180,E1 18868.289,E2 18868.289} C_VEL
LIN {X 0,Y 466.408,Z 565.05,A -85,B 0,C 180,E1 18865.232,E2 18865.232} C_VEL
LIN {X 0,Y 472.595,Z 578.951,A -85,B 0,C 180,E1 18862.303,E2 18862.303} C_VEL
LIN {X 0,Y 479.014,Z 594.767,A -85,B 0,C 180,E1 18859.363,E2 18859.363} C_VEL
LIN {X 0,Y 485.31,Z 611.995,A -85,B 0,C 180,E1 18856.516,E2 18856.516} C_VEL
LIN {X 0,Y 487.182,Z 617.951,A -85,B 0,C 180,E1 18855.62,E2 18855.62} C_VEL
LIN {X 0,Y 486.417,Z 623.852,A -85,B 0,C 180,E1 18855.143,E2 18855.143} C_VEL
LIN {X 0,Y 493.99,Z 674.926,A -85,B 0,C 180,E1 18853.139,E2 18853.139} C_VEL
LIN {X 0,Y 498.201,Z 706.483,A -85,B 0,C 180,E1 18852.034,E2 18852.034} C_VEL
LIN {X 0,Y 489.976,Z 950.582,A -85,B 0,C 180,E1 18848.514,E2 18848.514} C_VEL
LIN {X 0,Y 488.156,Z 972.978,A -85,B 0,C 180,E1 18848.029,E2 18848.029} C_VEL
LIN {X 0,Y 485.748,Z 994.344,A -85,B 0,C 180,E1 18847.385,E2 18847.385} C_VEL
LIN {X 0,Y 482.931,Z 1013.88,A -85,B 0,C 180,E1 18846.603,E2 18846.603} C_VEL
LIN {X 0,Y 479.262,Z 1035.34,A -85,B 0,C 180,E1 18845.529,E2 18845.529} C_VEL
LIN {X 0,Y 475.577,Z 1054.154,A -85,B 0,C 180,E1 18844.367,E2 18844.367} C_VEL
LIN {X 0,Y 471.406,Z 1073.012,A -85,B 0,C 180,E1 18842.959,E2 18842.959} C_VEL
LIN {X 0,Y 467.228,Z 1090.6,A -85,B 0,C 180,E1 18841.405,E2 18841.405} C_VEL
LIN {X 0,Y 462.83,Z 1107.558,A -85,B 0,C 180,E1 18839.609,E2 18839.609} C_VEL
LIN {X 0,Y 458.401,Z 1124.067,A -85,B 0,C 180,E1 18837.543,E2 18837.543} C_VEL
LIN {X 0,Y 454.444,Z 1138.541,A -85,B 0,C 180,E1 18835.406,E2 18835.406} C_VEL
LIN {X 0,Y 450.846,Z 1151.569,A -85,B 0,C 180,E1 18833.113,E2 18833.113} C_VEL
LIN {X 0,Y 447.553,Z 1163.969,A -85,B 0,C 180,E1 18830.533,E2 18830.533} C_VEL
LIN {X 0,Y 444.966,Z 1174.372,A -85,B 0,C 180,E1 18827.929,E2 18827.929} C_VEL
LIN {X 0,Y 442.945,Z 1183.347,A -85,B 0,C 180,E1 18825.18,E2 18825.18} C_VEL
LIN {X 0,Y 441.507,Z 1190.967,A -85,B 0,C 180,E1 18822.291,E2 18822.291} C_VEL
LIN {X 0,Y 440.991,Z 1194.266,A -85,B 0,C 180,E1 18820.776,E2 18820.776} C_VEL
LIN {X 0,Y 439.747,Z 1196.137,A -85,B 0,C 180,E1 18819.809,E2 18819.809} C_VEL
LIN {X 0,Y 432.905,Z 1200.582,A -85,B 0,C 180,E1 18817.147,E2 18817.147} C_VEL
LIN {X 0,Y 432.171,Z 1201.505,A -85,B 0,C 180,E1 18816.351,E2 18816.351} C_VEL
LIN {X 0,Y 432.004,Z 1204.094,A -85,B 0,C 180,E1 18813.317,E2 18813.317} C_VEL
LIN {X 0,Y 431.966,Z 1205.021,A -85,B 0,C 180,E1 18810.53,E2 18810.53} C_VEL
LIN {X 0,Y 431.986,Z 1204.525,A -85,B 0,C 180,E1 18807.48,E2 18807.48} C_VEL
LIN {X 0,Y 432.088,Z 1202.691,A -85,B 0,C 180,E1 18804.689,E2 18804.689} C_VEL
LIN {X 0,Y 432.401,Z 1199.23,A -85,B 0,C 180,E1 18801.757,E2 18801.757} C_VEL
LIN {X 0,Y 433.098,Z 1194.28,A -85,B 0,C 180,E1 18798.818,E2 18798.818} C_VEL
LIN {X 0,Y 434.304,Z 1187.518,A -85,B 0,C 180,E1 18795.875,E2 18795.875} C_VEL
LIN {X 0,Y 436.212,Z 1178.9,A -85,B 0,C 180,E1 18792.913,E2 18792.913} C_VEL
LIN {X 0,Y 438.716,Z 1169.036,A -85,B 0,C 180,E1 18790.149,E2 18790.149} C_VEL
LIN {X 0,Y 441.827,Z 1157.521,A -85,B 0,C 180,E1 18787.515,E2 18787.515} C_VEL
LIN {X 0,Y 445.484,Z 1144.648,A -85,B 0,C 180,E1 18785.042,E2 18785.042} C_VEL
LIN {X 0,Y 449.6,Z 1130.438,A -85,B 0,C 180,E1 18782.734,E2 18782.734} C_VEL
LIN {X 0,Y 453.914,Z 1115.083,A -85,B 0,C 180,E1 18780.652,E2 18780.652} C_VEL
LIN {X 0,Y 458.772,Z 1097.239,A -85,B 0,C 180,E1 18778.609,E2 18778.609} C_VEL
LIN {X 0,Y 463.33,Z 1079.592,A -85,B 0,C 180,E1 18776.909,E2 18776.909} C_VEL
LIN {X 0,Y 467.525,Z 1061.678,A -85,B 0,C 180,E1 18775.477,E2 18775.477} C_VEL
LIN {X 0,Y 471.624,Z 1042.55,A -85,B 0,C 180,E1 18774.188,E2 18774.188} C_VEL
LIN {X 0,Y 475.343,Z 1022.586,A -85,B 0,C 180,E1 18773.092,E2 18773.092} C_VEL
LIN {X 0,Y 478.72,Z 1001.165,A -85,B 0,C 180,E1 18772.151,E2 18772.151} C_VEL
LIN {X 0,Y 481.536,Z 979.543,A -85,B 0,C 180,E1 18771.418,E2 18771.418} C_VEL
LIN {X 0,Y 483.609,Z 957.374,A -85,B 0,C 180,E1 18770.888,E2 18770.888} C_VEL
LIN {X 0,Y 485.014,Z 928.059,A -85,B 0,C 180,E1 18770.407,E2 18770.407} C_VEL
LIN {X 0,Y 492.576,Z 706.156,A -85,B 0,C 180,E1 18767.181,E2 18767.181} C_VEL
LIN {X 0,Y 485.309,Z 653.444,A -85,B 0,C 180,E1 18765.207,E2 18765.207} C_VEL
LIN {X 0,Y 480.754,Z 621.616,A -85,B 0,C 180,E1 18763.877,E2 18763.877} C_VEL
LIN {X 0,Y 475.637,Z 606.583,A -85,B 0,C 180,E1 18761.468,E2 18761.468} C_VEL
LIN {X 0,Y 469.487,Z 590.595,A -85,B 0,C 180,E1 18758.594,E2 18758.594} C_VEL
LIN {X 0,Y 463.344,Z 576.008,A -85,B 0,C 180,E1 18755.638,E2 18755.638} C_VEL
LIN {X 0,Y 457.915,Z 564.272,A -85,B 0,C 180,E1 18752.937,E2 18752.937} C_VEL
LIN {X 0,Y 452.655,Z 553.183,A -85,B 0,C 180,E1 18750.095,E2 18750.095} C_VEL
LIN {X 0,Y 447.657,Z 543.585,A -85,B 0,C 180,E1 18747.251,E2 18747.251} C_VEL
LIN {X 0,Y 445.114,Z 538.841,A -85,B 0,C 180,E1 18745.693,E2 18745.693} C_VEL
LIN {X 0,Y 442.754,Z 534.34,A -85,B 0,C 180,E1 18744.127,E2 18744.127} C_VEL
LIN {X 0,Y 440.521,Z 530.186,A -85,B 0,C 180,E1 18742.557,E2 18742.557} C_VEL
LIN {X 0,Y 437.65,Z 525.317,A -85,B 0,C 180,E1 18740.46,E2 18740.46} C_VEL
LIN {X 0,Y 436.415,Z 523.455,A -85,B 0,C 180,E1 18739.543,E2 18739.543} C_VEL
LIN {X 0,Y 434.547,Z 519.904,A -85,B 0,C 180,E1 18737.82,E2 18737.82} C_VEL
LIN {X 0,Y 434.428,Z 519.157,A -85,B 0,C 180,E1 18737.227,E2 18737.227} C_VEL
LIN {X 0,Y 434.419,Z 519.097,A -85,B 0,C 180,E1 18733.443,E2 18733.443} C_VEL
LIN {X 0,Y 434.395,Z 519.088,A -85,B 0,C 180,E1 18729.673,E2 18729.673} C_VEL
LIN {X 0,Y 434.382,Z 519.085,A -85,B 0,C 180,E1 18725.946,E2 18725.946} C_VEL
LIN {X 0,Y 434.383,Z 519.093,A -85,B 0,C 180,E1 18722.111,E2 18722.111} C_VEL
LIN {X 0,Y 434.408,Z 519.113,A -85,B 0,C 180,E1 18718.417,E2 18718.417} C_VEL
LIN {X 0,Y 434.42,Z 519.11,A -85,B 0,C 180,E1 18714.585,E2 18714.585} C_VEL
LIN {X 0,Y 434.407,Z 519.091,A -85,B 0,C 180,E1 18710.862,E2 18710.862} C_VEL
LIN {X 0,Y 434.387,Z 519.087,A -85,B 0,C 180,E1 18707.098,E2 18707.098} C_VEL
LIN {X 0,Y 434.382,Z 519.132,A -85,B 0,C 180,E1 18703.415,E2 18703.415} C_VEL
LIN {X 0,Y 434.467,Z 519.55,A -85,B 0,C 180,E1 18702.729,E2 18702.729} C_VEL
LIN {X 0,Y 436.185,Z 523.263,A -85,B 0,C 180,E1 18701.003,E2 18701.003} C_VEL
LIN {X 0,Y 437.568,Z 524.882,A -85,B 0,C 180,E1 18700.094,E2 18700.094} C_VEL
LIN {X 0,Y 439.308,Z 528.515,A -85,B 0,C 180,E1 18698.643,E2 18698.643} C_VEL
LIN {X 0,Y 440.624,Z 530.43,A -85,B 0,C 180,E1 18697.793,E2 18697.793} C_VEL
LIN {X 0,Y 442.589,Z 534.07,A -85,B 0,C 180,E1 18696.429,E2 18696.429} C_VEL
LIN {X 0,Y 443.583,Z 535.873,A -85,B 0,C 180,E1 18695.779,E2 18695.779} C_VEL
LIN {X 0,Y 446.275,Z 540.835,A -85,B 0,C 180,E1 18694.093,E2 18694.093} C_VEL
LIN {X 0,Y 448.9,Z 545.772,A -85,B 0,C 180,E1 18692.543,E2 18692.543} C_VEL
LIN {X 0,Y 453.146,Z 553.718,A -85,B 0,C 180,E1 18690.233,E2 18690.233} C_VEL
LIN {X 0,Y 457.435,Z 562.176,A -85,B 0,C 180,E1 18688.1,E2 18688.1} C_VEL
LIN {X 0,Y 469.276,Z 577.732,A -85,B 0,C 180,E1 18685.697,E2 18685.697} C_VEL
LIN {X 0,Y 481.325,Z 594.589,A -85,B 0,C 180,E1 18683.475,E2 18683.475} C_VEL
LIN {X 0,Y 493.683,Z 613.44,A -85,B 0,C 180,E1 18681.367,E2 18681.367} C_VEL
LIN {X 0,Y 499.122,Z 622.732,A -85,B 0,C 180,E1 18680.477,E2 18680.477} C_VEL
LIN {X 0,Y 488.017,Z 860.617,A -85,B 0,C 180,E1 18676.62,E2 18676.62} C_VEL
LIN {X 0,Y 484.835,Z 927.115,A -85,B 0,C 180,E1 18675.503,E2 18675.503} C_VEL
LIN {X 0,Y 482.684,Z 951.547,A -85,B 0,C 180,E1 18674.905,E2 18674.905} C_VEL
LIN {X 0,Y 480.002,Z 975.456,A -85,B 0,C 180,E1 18674.127,E2 18674.127} C_VEL
LIN {X 0,Y 476.804,Z 998.036,A -85,B 0,C 180,E1 18673.171,E2 18673.171} C_VEL
LIN {X 0,Y 473.09,Z 1020.99,A -85,B 0,C 180,E1 18671.989,E2 18671.989} C_VEL
LIN {X 0,Y 469.229,Z 1041.651,A -85,B 0,C 180,E1 18670.696,E2 18670.696} C_VEL
LIN {X 0,Y 464.998,Z 1062.648,A -85,B 0,C 180,E1 18669.157,E2 18669.157} C_VEL
LIN {X 0,Y 460.593,Z 1082.48,A -85,B 0,C 180,E1 18667.432,E2 18667.432} C_VEL
LIN {X 0,Y 456.09,Z 1101.986,A -85,B 0,C 180,E1 18665.469,E2 18665.469} C_VEL
LIN {X 0,Y 451.918,Z 1119.292,A -85,B 0,C 180,E1 18663.429,E2 18663.429} C_VEL
LIN {X 0,Y 447.734,Z 1136.796,A -85,B 0,C 180,E1 18661.055,E2 18661.055} C_VEL
LIN {X 0,Y 444.076,Z 1151.96,A -85,B 0,C 180,E1 18658.658,E2 18658.658} C_VEL
LIN {X 0,Y 440.709,Z 1166.717,A -85,B 0,C 180,E1 18655.968,E2 18655.968} C_VEL
LIN {X 0,Y 438.101,Z 1178.776,A -85,B 0,C 180,E1 18653.398,E2 18653.398} C_VEL
LIN {X 0,Y 435.865,Z 1190.37,A -85,B 0,C 180,E1 18650.547,E2 18650.547} C_VEL
LIN {X 0,Y 434.225,Z 1200.036,A -85,B 0,C 180,E1 18647.695,E2 18647.695} C_VEL
LIN {X 0,Y 433.058,Z 1208.711,A -85,B 0,C 180,E1 18644.662,E2 18644.662} C_VEL
LIN {X 0,Y 432.383,Z 1215.282,A -85,B 0,C 180,E1 18641.741,E2 18641.741} C_VEL
LIN {X 0,Y 432.076,Z 1220.092,A -85,B 0,C 180,E1 18639.054,E2 18639.054} C_VEL
LIN {X 0,Y 431.947,Z 1224.194,A -85,B 0,C 180,E1 18635.846,E2 18635.846} C_VEL
LIN {X 0,Y 431.927,Z 1226.227,A -85,B 0,C 180,E1 18633.185,E2 18633.185} C_VEL
LIN {X 0,Y 431.929,Z 1227.073,A -85,B 0,C 180,E1 18630.663,E2 18630.663} C_VEL
LIN {X 0,Y 431.933,Z 1226.656,A -85,B 0,C 180,E1 18627.612,E2 18627.612} C_VEL
LIN {X 0,Y 431.926,Z 1224.911,A -85,B 0,C 180,E1 18624.953,E2 18624.953} C_VEL
LIN {X 0,Y 431.977,Z 1222.168,A -85,B 0,C 180,E1 18622.419,E2 18622.419} C_VEL
LIN {X 0,Y 432.212,Z 1217.674,A -85,B 0,C 180,E1 18619.47,E2 18619.47} C_VEL
LIN {X 0,Y 432.749,Z 1211.451,A -85,B 0,C 180,E1 18616.505,E2 18616.505} C_VEL
LIN {X 0,Y 433.639,Z 1204.113,A -85,B 0,C 180,E1 18613.662,E2 18613.662} C_VEL
LIN {X 0,Y 435.171,Z 1194.186,A -85,B 0,C 180,E1 18610.54,E2 18610.54} C_VEL
LIN {X 0,Y 437.058,Z 1183.947,A -85,B 0,C 180,E1 18607.823,E2 18607.823} C_VEL
LIN {X 0,Y 439.667,Z 1171.301,A -85,B 0,C 180,E1 18604.977,E2 18604.977} C_VEL
LIN {X 0,Y 442.478,Z 1158.809,A -85,B 0,C 180,E1 18602.55,E2 18602.55} C_VEL
LIN {X 0,Y 446.218,Z 1142.853,A -85,B 0,C 180,E1 18599.873,E2 18599.873} C_VEL
LIN {X 0,Y 449.855,Z 1127.772,A -85,B 0,C 180,E1 18597.687,E2 18597.687} C_VEL
LIN {X 0,Y 454.517,Z 1108.389,A -85,B 0,C 180,E1 18595.267,E2 18595.267} C_VEL
LIN {X 0,Y 458.611,Z 1090.986,A -85,B 0,C 180,E1 18593.396,E2 18593.396} C_VEL
LIN {X 0,Y 463.21,Z 1070.435,A -85,B 0,C 180,E1 18591.501,E2 18591.501} C_VEL
LIN {X 0,Y 467.278,Z 1051.24,A -85,B 0,C 180,E1 18589.985,E2 18589.985} C_VEL
LIN {X 0,Y 471.566,Z 1029.042,A -85,B 0,C 180,E1 18588.502,E2 18588.502} C_VEL
LIN {X 0,Y 474.967,Z 1009.468,A -85,B 0,C 180,E1 18587.4,E2 18587.4} C_VEL
LIN {X 0,Y 478.537,Z 985.826,A -85,B 0,C 180,E1 18586.299,E2 18586.299} C_VEL
LIN {X 0,Y 481.196,Z 964.898,A -85,B 0,C 180,E1 18585.517,E2 18585.517} C_VEL
LIN {X 0,Y 483.791,Z 939.545,A -85,B 0,C 180,E1 18584.79,E2 18584.79} C_VEL
LIN {X 0,Y 485.34,Z 917.456,A -85,B 0,C 180,E1 18584.329,E2 18584.329} C_VEL
LIN {X 0,Y 496.519,Z 675.655,A -85,B 0,C 180,E1 18580.378,E2 18580.378} C_VEL
LIN {X 0,Y 498.938,Z 622.164,A -85,B 0,C 180,E1 18579.506,E2 18579.506} C_VEL
LIN {X 0,Y 487.085,Z 603.194,A -85,B 0,C 180,E1 18577.548,E2 18577.548} C_VEL
LIN {X 0,Y 474.315,Z 584.621,A -85,B 0,C 180,E1 18575.283,E2 18575.283} C_VEL
LIN {X 0,Y 463.702,Z 570.464,A -85,B 0,C 180,E1 18573.247,E2 18573.247} C_VEL
LIN {X 0,Y 457.007,Z 561.615,A -85,B 0,C 180,E1 18571.822,E2 18571.822} C_VEL
LIN {X 0,Y 452.264,Z 552.298,A -85,B 0,C 180,E1 18569.394,E2 18569.394} C_VEL
LIN {X 0,Y 449.816,Z 547.658,A -85,B 0,C 180,E1 18568.06,E2 18568.06} C_VEL
LIN {X 0,Y 447.929,Z 543.892,A -85,B 0,C 180,E1 18566.946,E2 18566.946} C_VEL
LIN {X 0,Y 445.344,Z 539.057,A -85,B 0,C 180,E1 18565.394,E2 18565.394} C_VEL
LIN {X 0,Y 442.699,Z 534.198,A -85,B 0,C 180,E1 18563.706,E2 18563.706} C_VEL
LIN {X 0,Y 440.601,Z 530.381,A -85,B 0,C 180,E1 18562.271,E2 18562.271} C_VEL
LIN {X 0,Y 437.705,Z 525.406,A -85,B 0,C 180,E1 18560.178,E2 18560.178} C_VEL
LIN {X 0,Y 436.86,Z 523.952,A -85,B 0,C 180,E1 18559.522,E2 18559.522} C_VEL
LIN {X 0,Y 434.835,Z 520.849,A -85,B 0,C 180,E1 18557.947,E2 18557.947} C_VEL
LIN {X 0,Y 434.413,Z 519.232,A -85,B 0,C 180,E1 18557.135,E2 18557.135} C_VEL
LIN {X 0,Y 434.418,Z 519.089,A -85,B 0,C 180,E1 18553.443,E2 18553.443} C_VEL
LIN {X 0,Y 434.414,Z 519.101,A -85,B 0,C 180,E1 18549.673,E2 18549.673} C_VEL
LIN {X 0,Y 434.396,Z 519.118,A -85,B 0,C 180,E1 18545.945,E2 18545.945} C_VEL
LIN {X 0,Y 434.385,Z 519.098,A -85,B 0,C 180,E1 18542.111,E2 18542.111} C_VEL
LIN {X 0,Y 434.387,Z 519.086,A -85,B 0,C 180,E1 18538.285,E2 18538.285} C_VEL
LIN {X 0,Y 434.405,Z 519.084,A -85,B 0,C 180,E1 18534.585,E2 18534.585} C_VEL
LIN {X 0,Y 434.419,Z 519.094,A -85,B 0,C 180,E1 18530.862,E2 18530.862} C_VEL
LIN {X 0,Y 434.419,Z 519.109,A -85,B 0,C 180,E1 18526.964,E2 18526.964} C_VEL
LIN {X 0,Y 434.406,Z 519.116,A -85,B 0,C 180,E1 18523.234,E2 18523.234} C_VEL
LIN {X 0,Y 434.479,Z 519.573,A -85,B 0,C 180,E1 18522.107,E2 18522.107} C_VEL
LIN {X 0,Y 436.193,Z 523.2,A -85,B 0,C 180,E1 18520.408,E2 18520.408} C_VEL
LIN {X 0,Y 437.611,Z 525.176,A -85,B 0,C 180,E1 18519.398,E2 18519.398} C_VEL
LIN {X 0,Y 439.649,Z 528.956,A -85,B 0,C 180,E1 18517.819,E2 18517.819} C_VEL
LIN {X 0,Y 440.62,Z 530.491,A -85,B 0,C 180,E1 18517.167,E2 18517.167} C_VEL
LIN {X 0,Y 442.708,Z 534.291,A -85,B 0,C 180,E1 18515.728,E2 18515.728} C_VEL
LIN {X 0,Y 446.132,Z 540.737,A -85,B 0,C 180,E1 18513.512,E2 18513.512} C_VEL
LIN {X 0,Y 448.741,Z 545.809,A -85,B 0,C 180,E1 18511.926,E2 18511.926} C_VEL
LIN {X 0,Y 451.169,Z 550.577,A -85,B 0,C 180,E1 18510.528,E2 18510.528} C_VEL
LIN {X 0,Y 455.023,Z 558.059,A -85,B 0,C 180,E1 18508.467,E2 18508.467} C_VEL
LIN {X 0,Y 461.007,Z 570.897,A -85,B 0,C 180,E1 18505.371,E2 18505.371} C_VEL
LIN {X 0,Y 466.849,Z 584.186,A -85,B 0,C 180,E1 18502.535,E2 18502.535} C_VEL
LIN {X 0,Y 473.263,Z 600.239,A -85,B 0,C 180,E1 18499.514,E2 18499.514} C_VEL
LIN {X 0,Y 479.38,Z 617.295,A -85,B 0,C 180,E1 18496.667,E2 18496.667} C_VEL
LIN {X 0,Y 480.705,Z 621.583,A -85,B 0,C 180,E1 18496.027,E2 18496.027} C_VEL
LIN {X 0,Y 481.724,Z 629.782,A -85,B 0,C 180,E1 18495.655,E2 18495.655} C_VEL
LIN {X 0,Y 489.047,Z 680.615,A -85,B 0,C 180,E1 18493.643,E2 18493.643} C_VEL
LIN {X 0,Y 492.557,Z 707.973,A -85,B 0,C 180,E1 18492.677,E2 18492.677} C_VEL
LIN {X 0,Y 484.029,Z 950.334,A -85,B 0,C 180,E1 18489.148,E2 18489.148} C_VEL
LIN {X 0,Y 482.158,Z 972.699,A -85,B 0,C 180,E1 18488.66,E2 18488.66} C_VEL
LIN {X 0,Y 479.697,Z 993.937,A -85,B 0,C 180,E1 18488.019,E2 18488.019} C_VEL
LIN {X 0,Y 476.783,Z 1013.564,A -85,B 0,C 180,E1 18487.23,E2 18487.23} C_VEL
LIN {X 0,Y 473.177,Z 1034.172,A -85,B 0,C 180,E1 18486.2,E2 18486.2} C_VEL
LIN {X 0,Y 469.369,Z 1053.017,A -85,B 0,C 180,E1 18485.036,E2 18485.036} C_VEL
LIN {X 0,Y 464.875,Z 1072.803,A -85,B 0,C 180,E1 18483.556,E2 18483.556} C_VEL
LIN {X 0,Y 460.387,Z 1091.027,A -85,B 0,C 180,E1 18481.926,E2 18481.926} C_VEL
LIN {X 0,Y 455.929,Z 1107.631,A -85,B 0,C 180,E1 18480.146,E2 18480.146} C_VEL
LIN {X 0,Y 451.251,Z 1124.405,A -85,B 0,C 180,E1 18478.017,E2 18478.017} C_VEL
LIN {X 0,Y 447.15,Z 1138.859,A -85,B 0,C 180,E1 18475.851,E2 18475.851} C_VEL
LIN {X 0,Y 443.398,Z 1151.853,A -85,B 0,C 180,E1 18473.524,E2 18473.524} C_VEL
LIN {X 0,Y 439.962,Z 1164.228,A -85,B 0,C 180,E1 18470.904,E2 18470.904} C_VEL
LIN {X 0,Y 437.255,Z 1174.622,A -85,B 0,C 180,E1 18468.257,E2 18468.257} C_VEL
LIN {X 0,Y 435.129,Z 1183.58,A -85,B 0,C 180,E1 18465.459,E2 18465.459} C_VEL
LIN {X 0,Y 433.606,Z 1191.188,A -85,B 0,C 180,E1 18462.519,E2 18462.519} C_VEL
LIN {X 0,Y 432.719,Z 1196.766,A -85,B 0,C 180,E1 18459.711,E2 18459.711} C_VEL
LIN {X 0,Y 432.203,Z 1201.177,A -85,B 0,C 180,E1 18456.642,E2 18456.642} C_VEL
LIN {X 0,Y 432.171,Z 1201.505,A -85,B 0,C 180,E1 18456.351,E2 18456.351} C_VEL
LIN {X 0,Y 431.091,Z 1202.633,A -85,B 0,C 180,E1 18455.341,E2 18455.341} C_VEL
LIN {X 0,Y 424.632,Z 1204.799,A -85,B 0,C 180,E1 18452.559,E2 18452.559} C_VEL
LIN {X 0,Y 423.98,Z 1205.038,A -85,B 0,C 180,E1 18451.735,E2 18451.735} C_VEL
LIN {X 0,Y 423.971,Z 1205.156,A -85,B 0,C 180,E1 18448.919,E2 18448.919} C_VEL
LIN {X 0,Y 424.034,Z 1203.94,A -85,B 0,C 180,E1 18445.913,E2 18445.913} C_VEL
LIN {X 0,Y 424.229,Z 1201.349,A -85,B 0,C 180,E1 18443.096,E2 18443.096} C_VEL
LIN {X 0,Y 424.816,Z 1196.68,A -85,B 0,C 180,E1 18439.833,E2 18439.833} C_VEL
LIN {X 0,Y 425.858,Z 1190.756,A -85,B 0,C 180,E1 18436.836,E2 18436.836} C_VEL
LIN {X 0,Y 427.541,Z 1182.937,A -85,B 0,C 180,E1 18433.842,E2 18433.842} C_VEL
LIN {X 0,Y 429.99,Z 1173.253,A -85,B 0,C 180,E1 18430.861,E2 18430.861} C_VEL
LIN {X 0,Y 432.959,Z 1162.669,A -85,B 0,C 180,E1 18428.173,E2 18428.173} C_VEL
LIN {X 0,Y 436.454,Z 1150.596,A -85,B 0,C 180,E1 18425.647,E2 18425.647} C_VEL
LIN {X 0,Y 440.686,Z 1136.488,A -85,B 0,C 180,E1 18423.16,E2 18423.16} C_VEL
LIN {X 0,Y 445.072,Z 1121.783,A -85,B 0,C 180,E1 18420.972,E2 18420.972} C_VEL
LIN {X 0,Y 449.602,Z 1105.993,A -85,B 0,C 180,E1 18419.002,E2 18419.002} C_VEL
LIN {X 0,Y 454.396,Z 1088.554,A -85,B 0,C 180,E1 18417.153,E2 18417.153} C_VEL
LIN {X 0,Y 458.927,Z 1070.728,A -85,B 0,C 180,E1 18415.572,E2 18415.572} C_VEL
LIN {X 0,Y 463.413,Z 1051.349,A -85,B 0,C 180,E1 18414.141,E2 18414.141} C_VEL
LIN {X 0,Y 467.594,Z 1031.26,A -85,B 0,C 180,E1 18412.915,E2 18412.915} C_VEL
LIN {X 0,Y 471.1,Z 1011.195,A -85,B 0,C 180,E1 18411.935,E2 18411.935} C_VEL
LIN {X 0,Y 474.354,Z 988.967,A -85,B 0,C 180,E1 18411.079,E2 18411.079} C_VEL
LIN {X 0,Y 476.752,Z 968.215,A -85,B 0,C 180,E1 18410.483,E2 18410.483} C_VEL
LIN {X 0,Y 478.451,Z 945.527,A -85,B 0,C 180,E1 18410.026,E2 18410.026} C_VEL
LIN {X 0,Y 487.017,Z 707.624,A -85,B 0,C 180,E1 18406.523,E2 18406.523} C_VEL
LIN {X 0,Y 479.893,Z 654.802,A -85,B 0,C 180,E1 18404.507,E2 18404.507} C_VEL
LIN {X 0,Y 475.572,Z 625.596,A -85,B 0,C 180,E1 18403.269,E2 18403.269} C_VEL
LIN {X 0,Y 472.552,Z 619.818,A -85,B 0,C 180,E1 18402.618,E2 18402.618} C_VEL
LIN {X 0,Y 466.444,Z 602.809,A -85,B 0,C 180,E1 18399.687,E2 18399.687} C_VEL
LIN {X 0,Y 460.371,Z 587.649,A -85,B 0,C 180,E1 18396.735,E2 18396.735} C_VEL
LIN {X 0,Y 454.593,Z 574.373,A -85,B 0,C 180,E1 18393.813,E2 18393.813} C_VEL
LIN {X 0,Y 449.22,Z 562.882,A -85,B 0,C 180,E1 18390.942,E2 18390.942} C_VEL
LIN {X 0,Y 444.601,Z 553.698,A -85,B 0,C 180,E1 18388.329,E2 18388.329} C_VEL
LIN {X 0,Y 442.215,Z 549.072,A -85,B 0,C 180,E1 18386.886,E2 18386.886} C_VEL
LIN {X 0,Y 439.938,Z 544.733,A -85,B 0,C 180,E1 18385.44,E2 18385.44} C_VEL
LIN {X 0,Y 437.602,Z 540.287,A -85,B 0,C 180,E1 18383.856,E2 18383.856} C_VEL
LIN {X 0,Y 435.049,Z 535.527,A -85,B 0,C 180,E1 18382.002,E2 18382.002} C_VEL
LIN {X 0,Y 432.819,Z 531.541,A -85,B 0,C 180,E1 18380.275,E2 18380.275} C_VEL
LIN {X 0,Y 429.836,Z 526.426,A -85,B 0,C 180,E1 18377.742,E2 18377.742} C_VEL
LIN {X 0,Y 429.145,Z 525.152,A -85,B 0,C 180,E1 18377.072,E2 18377.072} C_VEL
LIN {X 0,Y 426.789,Z 521.538,A -85,B 0,C 180,E1 18374.795,E2 18374.795} C_VEL
LIN {X 0,Y 426.47,Z 520.202,A -85,B 0,C 180,E1 18373.836,E2 18373.836} C_VEL
LIN {X 0,Y 426.445,Z 520.075,A -85,B 0,C 180,E1 18369.992,E2 18369.992} C_VEL
LIN {X 0,Y 426.446,Z 520.074,A -85,B 0,C 180,E1 18366.192,E2 18366.192} C_VEL
LIN {X 0,Y 426.459,Z 520.084,A -85,B 0,C 180,E1 18362.419,E2 18362.419} C_VEL
LIN {X 0,Y 426.482,Z 520.107,A -85,B 0,C 180,E1 18358.657,E2 18358.657} C_VEL
LIN {X 0,Y 426.477,Z 520.093,A -85,B 0,C 180,E1 18354.754,E2 18354.754} C_VEL
LIN {X 0,Y 426.452,Z 520.078,A -85,B 0,C 180,E1 18351.098,E2 18351.098} C_VEL
LIN {X 0,Y 426.443,Z 520.089,A -85,B 0,C 180,E1 18347.257,E2 18347.257} C_VEL
LIN {X 0,Y 426.542,Z 520.499,A -85,B 0,C 180,E1 18346.166,E2 18346.166} C_VEL
LIN {X 0,Y 428.127,Z 524.038,A -85,B 0,C 180,E1 18344.142,E2 18344.142} C_VEL
LIN {X 0,Y 429.762,Z 526.064,A -85,B 0,C 180,E1 18342.814,E2 18342.814} C_VEL
LIN {X 0,Y 431.772,Z 529.998,A -85,B 0,C 180,E1 18340.942,E2 18340.942} C_VEL
LIN {X 0,Y 432.878,Z 531.52,A -85,B 0,C 180,E1 18340.15,E2 18340.15} C_VEL
LIN {X 0,Y 434.898,Z 535.292,A -85,B 0,C 180,E1 18338.558,E2 18338.558} C_VEL
LIN {X 0,Y 435.829,Z 536.877,A -85,B 0,C 180,E1 18337.898,E2 18337.898} C_VEL
LIN {X 0,Y 437.949,Z 540.604,A -85,B 0,C 180,E1 18336.45,E2 18336.45} C_VEL
LIN {X 0,Y 441.158,Z 546.662,A -85,B 0,C 180,E1 18334.348,E2 18334.348} C_VEL
LIN {X 0,Y 443.928,Z 552.068,A -85,B 0,C 180,E1 18332.646,E2 18332.646} C_VEL
LIN {X 0,Y 448.103,Z 560.088,A -85,B 0,C 180,E1 18330.306,E2 18330.306} C_VEL
LIN {X 0,Y 450.011,Z 563.591,A -85,B 0,C 180,E1 18329.415,E2 18329.415} C_VEL
LIN {X 0,Y 459.798,Z 576.299,A -85,B 0,C 180,E1 18327.289,E2 18327.289} C_VEL
LIN {X 0,Y 470.39,Z 590.525,A -85,B 0,C 180,E1 18325.198,E2 18325.198} C_VEL
LIN {X 0,Y 482.85,Z 608.788,A -85,B 0,C 180,E1 18322.924,E2 18322.924} C_VEL
LIN {X 0,Y 493.535,Z 626.011,A -85,B 0,C 180,E1 18321.107,E2 18321.107} C_VEL
LIN {X 0,Y 482.147,Z 862.413,A -85,B 0,C 180,E1 18317.246,E2 18317.246} C_VEL
LIN {X 0,Y 478.93,Z 927.485,A -85,B 0,C 180,E1 18316.144,E2 18316.144} C_VEL
LIN {X 0,Y 476.728,Z 951.775,A -85,B 0,C 180,E1 18315.545,E2 18315.545} C_VEL
LIN {X 0,Y 474.049,Z 975.036,A -85,B 0,C 180,E1 18314.786,E2 18314.786} C_VEL
LIN {X 0,Y 470.742,Z 997.755,A -85,B 0,C 180,E1 18313.822,E2 18313.822} C_VEL
LIN {X 0,Y 466.999,Z 1020.322,A -85,B 0,C 180,E1 18312.659,E2 18312.659} C_VEL
LIN {X 0,Y 462.824,Z 1041.906,A -85,B 0,C 180,E1 18311.299,E2 18311.299} C_VEL
LIN {X 0,Y 458.391,Z 1063.112,A -85,B 0,C 180,E1 18309.725,E2 18309.725} C_VEL
LIN {X 0,Y 454.05,Z 1081.988,A -85,B 0,C 180,E1 18308.067,E2 18308.067} C_VEL
LIN {X 0,Y 449.461,Z 1101.213,A -85,B 0,C 180,E1 18306.122,E2 18306.122} C_VEL
LIN {X 0,Y 444.922,Z 1119.238,A -85,B 0,C 180,E1 18303.976,E2 18303.976} C_VEL
LIN {X 0,Y 440.627,Z 1136.455,A -85,B 0,C 180,E1 18301.613,E2 18301.613} C_VEL
LIN {X 0,Y 436.797,Z 1151.636,A -85,B 0,C 180,E1 18299.181,E2 18299.181} C_VEL
LIN {X 0,Y 433.222,Z 1166.545,A -85,B 0,C 180,E1 18296.425,E2 18296.425} C_VEL
LIN {X 0,Y 430.372,Z 1179.095,A -85,B 0,C 180,E1 18293.698,E2 18293.698} C_VEL
LIN {X 0,Y 427.938,Z 1191.074,A -85,B 0,C 180,E1 18290.659,E2 18290.659} C_VEL
LIN {X 0,Y 426.323,Z 1200.214,A -85,B 0,C 180,E1 18287.893,E2 18287.893} C_VEL
LIN {X 0,Y 425.108,Z 1208.754,A -85,B 0,C 180,E1 18284.825,E2 18284.825} C_VEL
LIN {X 0,Y 424.397,Z 1215.327,A -85,B 0,C 180,E1 18281.828,E2 18281.828} C_VEL
LIN {X 0,Y 424.069,Z 1220.385,A -85,B 0,C 180,E1 18278.906,E2 18278.906} C_VEL
LIN {X 0,Y 423.946,Z 1224.107,A -85,B 0,C 180,E1 18275.821,E2 18275.821} C_VEL
LIN {X 0,Y 423.931,Z 1226.021,A -85,B 0,C 180,E1 18273.245,E2 18273.245} C_VEL
LIN {X 0,Y 423.932,Z 1226.869,A -85,B 0,C 180,E1 18270.676,E2 18270.676} C_VEL
LIN {X 0,Y 423.933,Z 1226.45,A -85,B 0,C 180,E1 18267.567,E2 18267.567} C_VEL
LIN {X 0,Y 423.926,Z 1224.703,A -85,B 0,C 180,E1 18264.858,E2 18264.858} C_VEL
LIN {X 0,Y 423.984,Z 1221.955,A -85,B 0,C 180,E1 18262.275,E2 18262.275} C_VEL
LIN {X 0,Y 424.238,Z 1217.453,A -85,B 0,C 180,E1 18259.27,E2 18259.27} C_VEL
LIN {X 0,Y 424.816,Z 1211.219,A -85,B 0,C 180,E1 18256.248,E2 18256.248} C_VEL
LIN {X 0,Y 425.767,Z 1203.874,A -85,B 0,C 180,E1 18253.351,E2 18253.351} C_VEL
LIN {X 0,Y 427.395,Z 1193.927,A -85,B 0,C 180,E1 18250.171,E2 18250.171} C_VEL
LIN {X 0,Y 429.406,Z 1183.678,A -85,B 0,C 180,E1 18247.406,E2 18247.406} C_VEL
LIN {X 0,Y 432.22,Z 1170.722,A -85,B 0,C 180,E1 18244.452,E2 18244.452} C_VEL
LIN {X 0,Y 435.328,Z 1157.643,A -85,B 0,C 180,E1 18241.885,E2 18241.885} C_VEL
LIN {X 0,Y 439.259,Z 1141.63,A -85,B 0,C 180,E1 18239.193,E2 18239.193} C_VEL
LIN {X 0,Y 443.359,Z 1125.492,A -85,B 0,C 180,E1 18236.847,E2 18236.847} C_VEL
LIN {X 0,Y 447.912,Z 1107.156,A -85,B 0,C 180,E1 18234.568,E2 18234.568} C_VEL
LIN {X 0,Y 452.614,Z 1088.01,A -85,B 0,C 180,E1 18232.512,E2 18232.512} C_VEL
LIN {X 0,Y 457.153,Z 1068.22,A -85,B 0,C 180,E1 18230.715,E2 18230.715} C_VEL
LIN {X 0,Y 461.742,Z 1047.23,A -85,B 0,C 180,E1 18229.078,E2 18229.078} C_VEL
LIN {X 0,Y 465.79,Z 1026.375,A -85,B 0,C 180,E1 18227.715,E2 18227.715} C_VEL
LIN {X 0,Y 469.707,Z 1004.227,A -85,B 0,C 180,E1 18226.495,E2 18226.495} C_VEL
LIN {X 0,Y 472.99,Z 982.185,A -85,B 0,C 180,E1 18225.512,E2 18225.512} C_VEL
LIN {X 0,Y 475.924,Z 959.356,A -85,B 0,C 180,E1 18224.689,E2 18224.689} C_VEL
LIN {X 0,Y 478.19,Z 935.745,A -85,B 0,C 180,E1 18224.054,E2 18224.054} C_VEL
LIN {X 0,Y 479.858,Z 910.486,A -85,B 0,C 180,E1 18223.557,E2 18223.557} C_VEL
LIN {X 0,Y 491.467,Z 666.256,A -85,B 0,C 180,E1 18219.549,E2 18219.549} C_VEL
LIN {X 0,Y 493.315,Z 625.655,A -85,B 0,C 180,E1 18218.877,E2 18218.877} C_VEL
LIN {X 0,Y 481.358,Z 606.605,A -85,B 0,C 180,E1 18216.837,E2 18216.837} C_VEL
LIN {X 0,Y 468.804,Z 588.252,A -85,B 0,C 180,E1 18214.528,E2 18214.528} C_VEL
LIN {X 0,Y 456.85,Z 572.382,A -85,B 0,C 180,E1 18212.13,E2 18212.13} C_VEL
LIN {X 0,Y 449.493,Z 562.907,A -85,B 0,C 180,E1 18210.477,E2 18210.477} C_VEL
LIN {X 0,Y 444.955,Z 554.069,A -85,B 0,C 180,E1 18208.012,E2 18208.012} C_VEL
LIN {X 0,Y 442.499,Z 549.406,A -85,B 0,C 180,E1 18206.578,E2 18206.578} C_VEL
LIN {X 0,Y 440.193,Z 544.978,A -85,B 0,C 180,E1 18205.136,E2 18205.136} C_VEL
LIN {X 0,Y 437.817,Z 540.451,A -85,B 0,C 180,E1 18203.557,E2 18203.557} C_VEL
LIN {X 0,Y 435.741,Z 536.64,A -85,B 0,C 180,E1 18202.107,E2 18202.107} C_VEL
LIN {X 0,Y 432.9,Z 531.645,A -85,B 0,C 180,E1 18199.989,E2 18199.989} C_VEL
LIN {X 0,Y 432.035,Z 530.255,A -85,B 0,C 180,E1 18199.327,E2 18199.327} C_VEL
LIN {X 0,Y 430.094,Z 527.084,A -85,B 0,C 180,E1 18197.731,E2 18197.731} C_VEL
LIN {X 0,Y 429.331,Z 525.369,A -85,B 0,C 180,E1 18196.925,E2 18196.925} C_VEL
LIN {X 0,Y 426.679,Z 521.267,A -85,B 0,C 180,E1 18194.383,E2 18194.383} C_VEL
LIN {X 0,Y 426.499,Z 520.197,A -85,B 0,C 180,E1 18193.697,E2 18193.697} C_VEL
LIN {X 0,Y 426.465,Z 520.095,A -85,B 0,C 180,E1 18189.855,E2 18189.855} C_VEL
LIN {X 0,Y 426.454,Z 520.103,A -85,B 0,C 180,E1 18186.057,E2 18186.057} C_VEL
LIN {X 0,Y 426.445,Z 520.083,A -85,B 0,C 180,E1 18182.284,E2 18182.284} C_VEL
LIN {X 0,Y 426.456,Z 520.072,A -85,B 0,C 180,E1 18178.522,E2 18178.522} C_VEL
LIN {X 0,Y 426.474,Z 520.072,A -85,B 0,C 180,E1 18174.754,E2 18174.754} C_VEL
LIN {X 0,Y 426.48,Z 520.084,A -85,B 0,C 180,E1 18170.962,E2 18170.962} C_VEL
LIN {X 0,Y 426.475,Z 520.102,A -85,B 0,C 180,E1 18167.13,E2 18167.13} C_VEL
LIN {X 0,Y 426.527,Z 520.546,A -85,B 0,C 180,E1 18165.5,E2 18165.5} C_VEL
LIN {X 0,Y 428.505,Z 524.517,A -85,B 0,C 180,E1 18163.181,E2 18163.181} C_VEL
LIN {X 0,Y 429.777,Z 526.257,A -85,B 0,C 180,E1 18162.115,E2 18162.115} C_VEL
LIN {X 0,Y 431.882,Z 530.087,A -85,B 0,C 180,E1 18160.244,E2 18160.244} C_VEL
LIN {X 0,Y 432.899,Z 531.77,A -85,B 0,C 180,E1 18159.446,E2 18159.446} C_VEL
LIN {X 0,Y 435.211,Z 535.7,A -85,B 0,C 180,E1 18157.723,E2 18157.723} C_VEL
LIN {X 0,Y 438.028,Z 540.799,A -85,B 0,C 180,E1 18155.739,E2 18155.739} C_VEL
LIN {X 0,Y 441.154,Z 547,A -85,B 0,C 180,E1 18153.625,E2 18153.625} C_VEL
LIN {X 0,Y 443.695,Z 551.984,A -85,B 0,C 180,E1 18152.047,E2 18152.047} C_VEL
LIN {X 0,Y 447.612,Z 559.507,A -85,B 0,C 180,E1 18149.821,E2 18149.821} C_VEL
LIN {X 0,Y 453.612,Z 572.239,A -85,B 0,C 180,E1 18146.559,E2 18146.559} C_VEL
LIN {X 0,Y 459.52,Z 585.644,A -85,B 0,C 180,E1 18143.556,E2 18143.556} C_VEL
LIN {X 0,Y 465.686,Z 600.963,A -85,B 0,C 180,E1 18140.539,E2 18140.539} C_VEL
LIN {X 0,Y 471.777,Z 617.645,A -85,B 0,C 180,E1 18137.625,E2 18137.625} C_VEL
LIN {X 0,Y 473.432,Z 621.89,A -85,B 0,C 180,E1 18137.006,E2 18137.006} C_VEL
LIN {X 0,Y 475.692,Z 626.311,A -85,B 0,C 180,E1 18136.579,E2 18136.579} C_VEL
LIN {X 0,Y 482.866,Z 677.074,A -85,B 0,C 180,E1 18134.511,E2 18134.511} C_VEL
LIN {X 0,Y 486.988,Z 709.226,A -85,B 0,C 180,E1 18133.338,E2 18133.338} C_VEL
LIN {X 0,Y 478.14,Z 950.068,A -85,B 0,C 180,E1 18129.798,E2 18129.798} C_VEL
LIN {X 0,Y 476.215,Z 972.468,A -85,B 0,C 180,E1 18129.306,E2 18129.306} C_VEL
LIN {X 0,Y 473.695,Z 993.59,A -85,B 0,C 180,E1 18128.666,E2 18128.666} C_VEL
LIN {X 0,Y 470.691,Z 1013.244,A -85,B 0,C 180,E1 18127.872,E2 18127.872} C_VEL
LIN {X 0,Y 466.977,Z 1033.895,A -85,B 0,C 180,E1 18126.835,E2 18126.835} C_VEL
LIN {X 0,Y 463.043,Z 1052.763,A -85,B 0,C 180,E1 18125.663,E2 18125.663} C_VEL
LIN {X 0,Y 458.396,Z 1072.587,A -85,B 0,C 180,E1 18124.171,E2 18124.171} C_VEL
LIN {X 0,Y 453.752,Z 1090.851,A -85,B 0,C 180,E1 18122.525,E2 18122.525} C_VEL
LIN {X 0,Y 449.132,Z 1107.478,A -85,B 0,C 180,E1 18120.725,E2 18120.725} C_VEL
LIN {X 0,Y 444.402,Z 1123.838,A -85,B 0,C 180,E1 18118.635,E2 18118.635} C_VEL
LIN {X 0,Y 440.113,Z 1138.355,A -85,B 0,C 180,E1 18116.441,E2 18116.441} C_VEL
LIN {X 0,Y 436.172,Z 1151.459,A -85,B 0,C 180,E1 18114.082,E2 18114.082} C_VEL
LIN {X 0,Y 432.721,Z 1163.381,A -85,B 0,C 180,E1 18111.555,E2 18111.555} C_VEL
LIN {X 0,Y 429.81,Z 1173.883,A -85,B 0,C 180,E1 18108.866,E2 18108.866} C_VEL
LIN {X 0,Y 427.413,Z 1183.426,A -85,B 0,C 180,E1 18105.885,E2 18105.885} C_VEL
LIN {X 0,Y 425.771,Z 1191.12,A -85,B 0,C 180,E1 18102.891,E2 18102.891} C_VEL
LIN {X 0,Y 424.805,Z 1196.741,A -85,B 0,C 180,E1 18100.031,E2 18100.031} C_VEL
LIN {X 0,Y 424.237,Z 1201.236,A -85,B 0,C 180,E1 18096.904,E2 18096.904} C_VEL
LIN {X 0,Y 424.036,Z 1203.883,A -85,B 0,C 180,E1 18094.056,E2 18094.056} C_VEL
LIN {X 0,Y 423.98,Z 1205.038,A -85,B 0,C 180,E1 18091.735,E2 18091.735} C_VEL
LIN {X 0,Y 422.973,Z 1205.233,A -85,B 0,C 180,E1 18090.694,E2 18090.694} C_VEL
LIN {X 0,Y 418.692,Z 1205.317,A -85,B 0,C 180,E1 18088.878,E2 18088.878} C_VEL
LIN {X 0,Y 416.26,Z 1204.999,A -85,B 0,C 180,E1 18087.534,E2 18087.534} C_VEL
LIN {X 0,Y 416,Z 1204.756,A -85,B 0,C 180,E1 18086.998,E2 18086.998} C_VEL
LIN {X 0,Y 416.154,Z 1202.61,A -85,B 0,C 180,E1 18083.932,E2 18083.932} C_VEL
LIN {X 0,Y 416.589,Z 1198.87,A -85,B 0,C 180,E1 18080.886,E2 18080.886} C_VEL
LIN {X 0,Y 417.509,Z 1193.279,A -85,B 0,C 180,E1 18077.694,E2 18077.694} C_VEL
LIN {X 0,Y 419.03,Z 1186.26,A -85,B 0,C 180,E1 18074.641,E2 18074.641} C_VEL
LIN {X 0,Y 421.169,Z 1177.698,A -85,B 0,C 180,E1 18071.738,E2 18071.738} C_VEL
LIN {X 0,Y 424.251,Z 1166.787,A -85,B 0,C 180,E1 18068.719,E2 18068.719} C_VEL
LIN {X 0,Y 427.863,Z 1154.929,A -85,B 0,C 180,E1 18066.008,E2 18066.008} C_VEL
LIN {X 0,Y 431.768,Z 1142.245,A -85,B 0,C 180,E1 18063.601,E2 18063.601} C_VEL
LIN {X 0,Y 436.352,Z 1127.509,A -85,B 0,C 180,E1 18061.237,E2 18061.237} C_VEL
LIN {X 0,Y 441.132,Z 1111.831,A -85,B 0,C 180,E1 18059.111,E2 18059.111} C_VEL
LIN {X 0,Y 445.905,Z 1095.256,A -85,B 0,C 180,E1 18057.235,E2 18057.235} C_VEL
LIN {X 0,Y 450.871,Z 1076.997,A -85,B 0,C 180,E1 18055.487,E2 18055.487} C_VEL
LIN {X 0,Y 455.203,Z 1059.58,A -85,B 0,C 180,E1 18054.093,E2 18054.093} C_VEL
LIN {X 0,Y 459.761,Z 1039.078,A -85,B 0,C 180,E1 18052.731,E2 18052.731} C_VEL
LIN {X 0,Y 463.798,Z 1018.54,A -85,B 0,C 180,E1 18051.62,E2 18051.62} C_VEL
LIN {X 0,Y 467.177,Z 997.528,A -85,B 0,C 180,E1 18050.731,E2 18050.731} C_VEL
LIN {X 0,Y 470.176,Z 974.426,A -85,B 0,C 180,E1 18049.988,E2 18049.988} C_VEL
LIN {X 0,Y 472.273,Z 952.133,A -85,B 0,C 180,E1 18049.475,E2 18049.475} C_VEL
LIN {X 0,Y 474.44,Z 897.77,A -85,B 0,C 180,E1 18048.646,E2 18048.646} C_VEL
LIN {X 0,Y 481.493,Z 708.902,A -85,B 0,C 180,E1 18045.842,E2 18045.842} C_VEL
LIN {X 0,Y 474.412,Z 655.006,A -85,B 0,C 180,E1 18043.744,E2 18043.744} C_VEL
LIN {X 0,Y 470.818,Z 630.088,A -85,B 0,C 180,E1 18042.669,E2 18042.669} C_VEL
LIN {X 0,Y 464.636,Z 619.07,A -85,B 0,C 180,E1 18041.433,E2 18041.433} C_VEL
LIN {X 0,Y 458.781,Z 603.197,A -85,B 0,C 180,E1 18038.559,E2 18038.559} C_VEL
LIN {X 0,Y 452.765,Z 588.31,A -85,B 0,C 180,E1 18035.508,E2 18035.508} C_VEL
LIN {X 0,Y 447.23,Z 575.897,A -85,B 0,C 180,E1 18032.603,E2 18032.603} C_VEL
LIN {X 0,Y 442.1,Z 564.841,A -85,B 0,C 180,E1 18029.69,E2 18029.69} C_VEL
LIN {X 0,Y 437.485,Z 555.664,A -85,B 0,C 180,E1 18026.907,E2 18026.907} C_VEL
LIN {X 0,Y 434.779,Z 550.61,A -85,B 0,C 180,E1 18025.18,E2 18025.18} C_VEL
LIN {X 0,Y 432.693,Z 546.515,A -85,B 0,C 180,E1 18023.709,E2 18023.709} C_VEL
LIN {X 0,Y 430.166,Z 541.778,A -85,B 0,C 180,E1 18021.834,E2 18021.834} C_VEL
LIN {X 0,Y 427.883,Z 537.394,A -85,B 0,C 180,E1 18019.949,E2 18019.949} C_VEL
LIN {X 0,Y 425.276,Z 533.279,A -85,B 0,C 180,E1 18017.79,E2 18017.79} C_VEL
LIN {X 0,Y 424.523,Z 531.658,A -85,B 0,C 180,E1 18016.981,E2 18016.981} C_VEL
LIN {X 0,Y 422.202,Z 528.043,A -85,B 0,C 180,E1 18014.679,E2 18014.679} C_VEL
LIN {X 0,Y 421.367,Z 526.308,A -85,B 0,C 180,E1 18013.587,E2 18013.587} C_VEL
LIN {X 0,Y 418.629,Z 521.725,A -85,B 0,C 180,E1 18009.625,E2 18009.625} C_VEL
LIN {X 0,Y 418.517,Z 521.138,A -85,B 0,C 180,E1 18008.242,E2 18008.242} C_VEL
LIN {X 0,Y 418.519,Z 521.075,A -85,B 0,C 180,E1 18004.385,E2 18004.385} C_VEL
LIN {X 0,Y 418.538,Z 521.059,A -85,B 0,C 180,E1 18000.548,E2 18000.548} C_VEL
LIN {X 0,Y 418.535,Z 521.058,A -85,B 0,C 180,E1 17996.713,E2 17996.713} C_VEL
LIN {X 0,Y 418.537,Z 521.065,A -85,B 0,C 180,E1 17992.864,E2 17992.864} C_VEL
LIN {X 0,Y 418.596,Z 521.534,A -85,B 0,C 180,E1 17990.929,E2 17990.929} C_VEL
LIN {X 0,Y 421.22,Z 526.176,A -85,B 0,C 180,E1 17986.967,E2 17986.967} C_VEL
LIN {X 0,Y 421.957,Z 527.263,A -85,B 0,C 180,E1 17986.153,E2 17986.153} C_VEL
LIN {X 0,Y 424.024,Z 531.14,A -85,B 0,C 180,E1 17983.844,E2 17983.844} C_VEL
LIN {X 0,Y 425.142,Z 532.623,A -85,B 0,C 180,E1 17982.903,E2 17982.903} C_VEL
LIN {X 0,Y 427.161,Z 536.514,A -85,B 0,C 180,E1 17981.012,E2 17981.012} C_VEL
LIN {X 0,Y 428.18,Z 538.082,A -85,B 0,C 180,E1 17980.23,E2 17980.23} C_VEL
LIN {X 0,Y 430.269,Z 541.813,A -85,B 0,C 180,E1 17978.602,E2 17978.602} C_VEL
LIN {X 0,Y 433.626,Z 547.978,A -85,B 0,C 180,E1 17976.201,E2 17976.201} C_VEL
LIN {X 0,Y 436.399,Z 553.392,A -85,B 0,C 180,E1 17974.339,E2 17974.339} C_VEL
LIN {X 0,Y 438.961,Z 558.352,A -85,B 0,C 180,E1 17972.751,E2 17972.751} C_VEL
LIN {X 0,Y 442.455,Z 564.877,A -85,B 0,C 180,E1 17970.856,E2 17970.856} C_VEL
LIN {X 0,Y 452.408,Z 577.451,A -85,B 0,C 180,E1 17968.56,E2 17968.56} C_VEL
LIN {X 0,Y 462.55,Z 591.002,A -85,B 0,C 180,E1 17966.437,E2 17966.437} C_VEL
LIN {X 0,Y 473.745,Z 606.993,A -85,B 0,C 180,E1 17964.278,E2 17964.278} C_VEL
LIN {X 0,Y 485.497,Z 625.339,A -85,B 0,C 180,E1 17962.177,E2 17962.177} C_VEL
LIN {X 0,Y 487.985,Z 629.875,A -85,B 0,C 180,E1 17961.741,E2 17961.741} C_VEL
LIN {X 0,Y 476.242,Z 866.204,A -85,B 0,C 180,E1 17957.854,E2 17957.854} C_VEL
LIN {X 0,Y 473.078,Z 928.023,A -85,B 0,C 180,E1 17956.797,E2 17956.797} C_VEL
LIN {X 0,Y 470.799,Z 952.335,A -85,B 0,C 180,E1 17956.191,E2 17956.191} C_VEL
LIN {X 0,Y 467.947,Z 976.164,A -85,B 0,C 180,E1 17955.402,E2 17955.402} C_VEL
LIN {X 0,Y 464.551,Z 998.699,A -85,B 0,C 180,E1 17954.432,E2 17954.432} C_VEL
LIN {X 0,Y 460.559,Z 1021.745,A -85,B 0,C 180,E1 17953.221,E2 17953.221} C_VEL
LIN {X 0,Y 456.472,Z 1042.168,A -85,B 0,C 180,E1 17951.918,E2 17951.918} C_VEL
LIN {X 0,Y 451.823,Z 1063.607,A -85,B 0,C 180,E1 17950.307,E2 17950.307} C_VEL
LIN {X 0,Y 447.233,Z 1082.871,A -85,B 0,C 180,E1 17948.59,E2 17948.59} C_VEL
LIN {X 0,Y 442.329,Z 1102.514,A -85,B 0,C 180,E1 17946.557,E2 17946.557} C_VEL
LIN {X 0,Y 437.83,Z 1119.742,A -85,B 0,C 180,E1 17944.469,E2 17944.469} C_VEL
LIN {X 0,Y 433.088,Z 1137.866,A -85,B 0,C 180,E1 17941.917,E2 17941.917} C_VEL
LIN {X 0,Y 429.353,Z 1152.115,A -85,B 0,C 180,E1 17939.584,E2 17939.584} C_VEL
LIN {X 0,Y 425.488,Z 1167.459,A -85,B 0,C 180,E1 17936.669,E2 17936.669} C_VEL
LIN {X 0,Y 422.656,Z 1179.417,A -85,B 0,C 180,E1 17934.01,E2 17934.01} C_VEL
LIN {X 0,Y 420.013,Z 1191.781,A -85,B 0,C 180,E1 17930.775,E2 17930.775} C_VEL
LIN {X 0,Y 418.355,Z 1200.819,A -85,B 0,C 180,E1 17927.957,E2 17927.957} C_VEL
LIN {X 0,Y 417.033,Z 1209.734,A -85,B 0,C 180,E1 17924.581,E2 17924.581} C_VEL
LIN {X 0,Y 416.388,Z 1215.641,A -85,B 0,C 180,E1 17921.777,E2 17921.777} C_VEL
LIN {X 0,Y 416.057,Z 1220.906,A -85,B 0,C 180,E1 17918.569,E2 17918.569} C_VEL
LIN {X 0,Y 415.935,Z 1224.197,A -85,B 0,C 180,E1 17915.591,E2 17915.591} C_VEL
LIN {X 0,Y 415.927,Z 1225.96,A -85,B 0,C 180,E1 17913.032,E2 17913.032} C_VEL
LIN {X 0,Y 415.955,Z 1226.776,A -85,B 0,C 180,E1 17910,E2 17910} C_VEL
LIN {X 0,Y 415.927,Z 1225.956,A -85,B 0,C 180,E1 17906.968,E2 17906.968} C_VEL
LIN {X 0,Y 415.938,Z 1224.132,A -85,B 0,C 180,E1 17904.344,E2 17904.344} C_VEL
LIN {X 0,Y 416.063,Z 1220.724,A -85,B 0,C 180,E1 17901.292,E2 17901.292} C_VEL
LIN {X 0,Y 416.388,Z 1215.626,A -85,B 0,C 180,E1 17898.223,E2 17898.223} C_VEL
LIN {X 0,Y 417.031,Z 1209.713,A -85,B 0,C 180,E1 17895.419,E2 17895.419} C_VEL
LIN {X 0,Y 418.358,Z 1200.763,A -85,B 0,C 180,E1 17892.034,E2 17892.034} C_VEL
LIN {X 0,Y 420.01,Z 1191.752,A -85,B 0,C 180,E1 17889.225,E2 17889.225} C_VEL
LIN {X 0,Y 422.653,Z 1179.379,A -85,B 0,C 180,E1 17885.99,E2 17885.99} C_VEL
LIN {X 0,Y 425.482,Z 1167.411,A -85,B 0,C 180,E1 17883.331,E2 17883.331} C_VEL
LIN {X 0,Y 429.343,Z 1152.049,A -85,B 0,C 180,E1 17880.416,E2 17880.416} C_VEL
LIN {X 0,Y 433.08,Z 1137.791,A -85,B 0,C 180,E1 17878.083,E2 17878.083} C_VEL
LIN {X 0,Y 437.595,Z 1120.513,A -85,B 0,C 180,E1 17875.642,E2 17875.642} C_VEL
LIN {X 0,Y 442.006,Z 1103.546,A -85,B 0,C 180,E1 17873.573,E2 17873.573} C_VEL
LIN {X 0,Y 447.05,Z 1083.414,A -85,B 0,C 180,E1 17871.473,E2 17871.473} C_VEL
LIN {X 0,Y 451.512,Z 1064.674,A -85,B 0,C 180,E1 17869.796,E2 17869.796} C_VEL
LIN {X 0,Y 456.267,Z 1042.894,A -85,B 0,C 180,E1 17868.143,E2 17868.143} C_VEL
LIN {X 0,Y 460.36,Z 1022.432,A -85,B 0,C 180,E1 17866.831,E2 17866.831} C_VEL
LIN {X 0,Y 464.419,Z 999.098,A -85,B 0,C 180,E1 17865.597,E2 17865.597} C_VEL
LIN {X 0,Y 467.815,Z 976.574,A -85,B 0,C 180,E1 17864.625,E2 17864.625} C_VEL
LIN {X 0,Y 470.709,Z 952.482,A -85,B 0,C 180,E1 17863.823,E2 17863.823} C_VEL
LIN {X 0,Y 472.99,Z 928.185,A -85,B 0,C 180,E1 17863.216,E2 17863.216} C_VEL
LIN {X 0,Y 476.214,Z 865.219,A -85,B 0,C 180,E1 17862.139,E2 17862.139} C_VEL
LIN {X 0,Y 487.905,Z 629.646,A -85,B 0,C 180,E1 17858.265,E2 17858.265} C_VEL
LIN {X 0,Y 478.475,Z 614.234,A -85,B 0,C 180,E1 17856.61,E2 17856.61} C_VEL
LIN {X 0,Y 466.543,Z 596.559,A -85,B 0,C 180,E1 17854.384,E2 17854.384} C_VEL
LIN {X 0,Y 454.176,Z 579.676,A -85,B 0,C 180,E1 17851.859,E2 17851.859} C_VEL
LIN {X 0,Y 445.35,Z 568.636,A -85,B 0,C 180,E1 17849.896,E2 17849.896} C_VEL
LIN {X 0,Y 442.118,Z 564.447,A -85,B 0,C 180,E1 17849.094,E2 17849.094} C_VEL
LIN {X 0,Y 437.812,Z 556.013,A -85,B 0,C 180,E1 17846.592,E2 17846.592} C_VEL
LIN {X 0,Y 435.287,Z 551.215,A -85,B 0,C 180,E1 17845.003,E2 17845.003} C_VEL
LIN {X 0,Y 432.707,Z 546.412,A -85,B 0,C 180,E1 17843.275,E2 17843.275} C_VEL
LIN {X 0,Y 430.129,Z 541.653,A -85,B 0,C 180,E1 17841.406,E2 17841.406} C_VEL
LIN {X 0,Y 428.031,Z 537.659,A -85,B 0,C 180,E1 17839.715,E2 17839.715} C_VEL
LIN {X 0,Y 425.357,Z 533.318,A -85,B 0,C 180,E1 17837.511,E2 17837.511} C_VEL
LIN {X 0,Y 424.547,Z 531.71,A -85,B 0,C 180,E1 17836.698,E2 17836.698} C_VEL
LIN {X 0,Y 422.013,Z 527.505,A -85,B 0,C 180,E1 17834.125,E2 17834.125} C_VEL
LIN {X 0,Y 421.344,Z 526.254,A -85,B 0,C 180,E1 17833.308,E2 17833.308} C_VEL
LIN {X 0,Y 418.68,Z 521.884,A -85,B 0,C 180,E1 17829.624,E2 17829.624} C_VEL
LIN {X 0,Y 418.512,Z 521.14,A -85,B 0,C 180,E1 17828.38,E2 17828.38} C_VEL
LIN {X 0,Y 418.509,Z 521.066,A -85,B 0,C 180,E1 17824.522,E2 17824.522} C_VEL
LIN {X 0,Y 418.525,Z 521.084,A -85,B 0,C 180,E1 17820.684,E2 17820.684} C_VEL
LIN {X 0,Y 418.536,Z 521.088,A -85,B 0,C 180,E1 17816.85,E2 17816.85} C_VEL
LIN {X 0,Y 418.547,Z 521.069,A -85,B 0,C 180,E1 17812.864,E2 17812.864} C_VEL
LIN {X 0,Y 418.581,Z 521.495,A -85,B 0,C 180,E1 17810.201,E2 17810.201} C_VEL
LIN {X 0,Y 421.23,Z 526.181,A -85,B 0,C 180,E1 17806.268,E2 17806.268} C_VEL
LIN {X 0,Y 422.136,Z 527.826,A -85,B 0,C 180,E1 17805.178,E2 17805.178} C_VEL
LIN {X 0,Y 424.236,Z 531.381,A -85,B 0,C 180,E1 17803.007,E2 17803.007} C_VEL
LIN {X 0,Y 425.119,Z 532.809,A -85,B 0,C 180,E1 17802.196,E2 17802.196} C_VEL
LIN {X 0,Y 427.431,Z 536.811,A -85,B 0,C 180,E1 17800.172,E2 17800.172} C_VEL
LIN {X 0,Y 430.86,Z 543.051,A -85,B 0,C 180,E1 17797.458,E2 17797.458} C_VEL
LIN {X 0,Y 433.594,Z 548.274,A -85,B 0,C 180,E1 17795.475,E2 17795.475} C_VEL
LIN {X 0,Y 436.333,Z 553.595,A -85,B 0,C 180,E1 17793.634,E2 17793.634} C_VEL
LIN {X 0,Y 440.268,Z 561.14,A -85,B 0,C 180,E1 17791.236,E2 17791.236} C_VEL
LIN {X 0,Y 446.08,Z 573.244,A -85,B 0,C 180,E1 17787.911,E2 17787.911} C_VEL
LIN {X 0,Y 451.761,Z 586.043,A -85,B 0,C 180,E1 17784.868,E2 17784.868} C_VEL
LIN {X 0,Y 457.649,Z 600.439,A -85,B 0,C 180,E1 17781.861,E2 17781.861} C_VEL
LIN {X 0,Y 463.333,Z 615.588,A -85,B 0,C 180,E1 17779.05,E2 17779.05} C_VEL
LIN {X 0,Y 465.237,Z 620.423,A -85,B 0,C 180,E1 17778.283,E2 17778.283} C_VEL
LIN {X 0,Y 470.891,Z 630.635,A -85,B 0,C 180,E1 17777.186,E2 17777.186} C_VEL
LIN {X 0,Y 477.928,Z 681.978,A -85,B 0,C 180,E1 17775.071,E2 17775.071} C_VEL
